// TwinCAT 3 PLC project SlaveController
// ProgramVersion: 3.1.4024.0
// libraries:
//   Tc2_EtherCAT, * (Beckhoff Automation GmbH)
//   Tc2_Math, * (Beckhoff Automation GmbH)
//   Tc2_Standard, * (Beckhoff Automation GmbH)
//   Tc2_System, * (Beckhoff Automation GmbH)
//   Tc2_Utilities, * (Beckhoff Automation GmbH)
//   Tc3_Module, * (Beckhoff Automation GmbH)
// project tree:
//   AgiMaths/Frames/ DHTrans.TcPOU (not stored), invFrame.TcPOU (not stored), rotX.TcPOU (not stored), rotY.TcPOU (not stored), rotZ.TcPOU (not stored), transform.TcPOU (not stored)
//   AgiMaths/MatrixLib/ angAxis2Rot.TcPOU (not stored), cross.TcPOU (not stored), Det5.TcPOU (not stored), Det6.TcPOU (not stored), Det7.TcPOU (not stored), invMat6.TcPOU (not stored), invMat6Old.TcPOU (not stored), invMat3.TcPOU (not stored), invMat7.TcPOU (not stored), Mat3T.TcPOU (not stored), matAdd.TcPOU (not stored), matMultiNum.TcPOU (not stored), matMultiply.TcPOU (not stored), matMultiVec.TcPOU (not stored), matSelfAdd.TcPOU (not stored), vecSelfAdd.TcPOU (not stored), matSelfSub.TcPOU (not stored), matSub.TcPOU (not stored), matTranspose.TcPOU (not stored), rot2AngAxis.TcPOU (not stored), vecAdd.TcPOU (not stored), norm.TcPOU (not stored), normalize.TcPOU (not stored), vecSelfMultiNum.TcPOU (not stored), vecMultiNum.TcPOU (not stored), vecSub.TcPOU (not stored)
//   AgiMaths/ sign.TcPOU (not stored), addVec7.TcPOU (not stored), atan2.TcPOU (not stored), cot.TcPOU (not stored)
//   DUTs/Enum/ E_CartJointState.TcTLEO (not stored), E_InstrumentType.TcDUT, E_MasterArmState.TcDUT (not stored), E_MatchedSlaveArmIdx.TcDUT (not stored), E_SetupArmState.TcDUT (not stored), E_SlaveArmState.TcDUT, E_DriverCtrlWord.TcDUT (not stored), E_DriverOPMode.TcDUT (not stored), E_DriverStatusWord.TcDUT
//   DUTs/Structure/MasterSlaveCommunication/ ST_MasterStatus.TcDUT, ST_SlaveStatus.TcDUT
//   DUTs/Structure/ ST_CartInputDataPool.TcDUT, ST_InstruOnChipData.TcDUT (not stored), ST_InstruStatus.TcDUT (not stored), ST_SetupArmCtrlCmds.TcDUT, ST_SetupInputDataPool.TcDUT, ST_SlaveArmCtrlCmds.TcDUT (not stored), ST_SlaveInputDataPool.TcDUT (not stored), ST_InstruKinematicParam.TcDUT, ST_Frame.TcDUT (not stored)
//   DUTs/Structure/TasksCommunication/ ST_CartJointData.TcDUT (not stored), ST_CartMotorInput.TcDUT (not stored), ST_CartMotorOutput.TcDUT (not stored), ST_CartUIData.TcDUT (not stored), ST_SetupStatus.TcDUT (not stored), ST_SetupJointData.TcDUT (not stored), ST_SlaveDynaData.TcDUT (not stored), ST_SlaveUIData.TcDUT (not stored), ST_CartStatus.TcDUT (not stored), ST_MasterJointData.TcDUT (not stored), ST_MotorInputs.TcDUT (not stored), ST_MotorOutputs.TcDUT (not stored), ST_SlaveJointData.TcDUT (not stored), ST_SafetyData.TcDUT
//   DUTs/Structure/UICommunication/ ST_cart_operation.TcDUT, ST_DH.TcDUT (not stored), ST_instrument_info.TcDUT (not stored), ST_scope_info.TcDUT, ST_state_machine_com.TcDUT (not stored), ST_ui_control.TcDUT (not stored)
//   DUTs/Type/ Mat34.TcDUT (not stored), Mat37.TcDUT (not stored), Mat43.TcDUT (not stored), Mat45.TcDUT (not stored), Mat4d.TcDUT (not stored), Mat5d.TcDUT (not stored), Mat67.TcDUT (not stored), Mat6d.TcDUT (not stored), Mat76.TcDUT (not stored), Mat7d.TcDUT (not stored), Vec2i.TcDUT, Vec4b.TcDUT (not stored), Vec4d.TcDUT (not stored), Vec4i.TcDUT (not stored), Vec5b.TcDUT (not stored), Vec5d.TcDUT (not stored), Vec5i.TcDUT (not stored), Vec6i.TcDUT (not stored), Vec8b.TcDUT (not stored), Vec8d.TcDUT (not stored), Vec8i.TcDUT (not stored), Mat3d.TcDUT (not stored), Vec3d.TcDUT (not stored), Vec6d.TcDUT (not stored), Vec7d.TcDUT (not stored), Vec7i.TcDUT (not stored)
//   FBs_Auxiliary/ FB_IOCheck.TcPOU (not stored), FB_IOToggleCheck.TcPOU (not stored), FB_rotaButtonDetect.TcPOU (not stored), FB_setupAdjustDetect.TcPOU, FB_setupJnt5AdjustDetect.TcPOU (not stored), FB_masterConnectionCheck.TcPOU (not stored), FB_trocarCheckDetect.TcPOU (not stored), FB_TrocarDetect.TcPOU, FB_PanelDetect.TcPOU, FB_InstrumentDetect.TcPOU, FB_AdjustDetect.TcPOU (not stored)
//   FBs_BasicControllers/ FB_dither.TcPOU (not stored), FB_InstrumentControl.TcPOU (not stored), FBMacroJntControl.TcPOU (not stored), FB_PID.TcPOU (not stored)
//   FBs_CartControlles/ FB_CartCtrlAdjust.TcPOU (not stored), FB_CartCtrlAsepticDeploy.TcPOU, FB_CartCtrlBase.TcPOU, FB_CartCtrlError.TcPOU, FB_CartCtrlInit.TcPOU (not stored), FB_CartCtrlInSurgery.TcPOU (not stored), FB_CartCtrlMotionCar.TcPOU (not stored), FB_CartCtrlReady.TcPOU, FB_CartCtrlRotaOverhang.TcPOU, FB_CartCtrlSlowDown.TcPOU, I_CartJointCtrl.TcIO
//   FBs_RobotDynamics/ FB_SlaveGravity.TcPOU, FB_SetupGravity.TcPOU
//   FBs_Robots/ FB_CartJoint.TcPOU (not stored), FB_CartRobot.TcPOU, FB_Instrument.TcPOU, FB_JointBase.TcPOU (not stored), FB_SlaveCart.TcPOU (not stored), FB_SetupArm.TcPOU (not stored), FB_SlaveJoint.TcPOU, FB_SetupJoint.TcPOU (not stored), FB_SetupRobot.TcPOU (not stored), FB_SlaveArm.TcPOU (not stored), FB_SlaveRobot.TcPOU (not stored)
//   FBs_SetupControllers/ FB_SetupCtrlDisable.TcPOU (not stored), FB_SetupCtrlJnt5GraCali.TcPOU, FB_SetupCtrlHold.TcPOU (not stored), FB_SetupCtrlManualAdjust.TcPOU, FB_SetupArmCtrlBase.TcPOU (not stored), FB_SetupCtrlAutoAdjust.TcPOU (not stored), FB_SetupCtrlCart.TcPOU (not stored), FB_SetupCtrlError.TcPOU (not stored), FB_SetupCtrlJnt3GraCali.TcPOU (not stored), FB_SetupCtrlInit.TcPOU (not stored), FB_SetupCtrlPackage.TcPOU (not stored), FB_SetupCtrlSelfCheck.TcPOU (not stored), I_SetupArmCtrl.TcIO (not stored)
//   FBs_SlaveControllers/ FB_SlaveCtrlDisable.TcPOU (not stored), FB_SlaveCtrlInstruInvasion.TcPOU, FB_SlaveCtrlInstruRetract.TcPOU (not stored), FB_SlaveCtrlInstruCali.TcPOU, FB_SlaveCtrlTest.TcPOU (not stored), FB_SlaveCtrlPackage.TcPOU (not stored), FB_SlaveCtrlEndoscope.TcPOU (not stored), FB_SlaveCtrlCart.TcPOU (not stored), FB_SlaveCtrlScopeReady.TcPOU (not stored), FB_SlaveCtrlSelfCheck.TcPOU (not stored), FB_SlaveCtrlError.TcPOU, FB_SlaveCtrlInstruReady.TcPOU (not stored), FB_SlaveCtrlMasterSlave.TcPOU (not stored), FB_SlaveCtrlMountInstru.TcPOU, FB_SlaveCtrlAdjust.TcPOU, FB_SlaveCtrlMountPanel.TcPOU (not stored), FB_SlaveCtrlPanelReady.TcPOU (not stored), FB_SlaveCtrlGraCali.TcPOU, FB_SlaveCtrlInit.TcPOU (not stored), FB_SlaveCtrlStandBy.TcPOU (not stored), FB_SlaveArmCtrlBase.TcPOU (not stored), I_SlaveArmCtrl.TcIO (not stored)
//   FBs_TrajectoryPlanning/ FB_BasicDoubleS.TcPOU (not stored), FB_trajBase.TcPOU (not stored), FB_TrajMoveJ.TcPOU (not stored), FB_setupTrajMoveJ.TcPOU (not stored), linear_trajectory_with_quintic_polynomial_blends.TcPOU (not stored), quintic_spline_curve.TcPOU (not stored), Quintic_spline_curve_factor.TcPOU (not stored), TrapezoIDal_velocity_trajectory.TcPOU (not stored)
//   FBs_TrajectoryPlanning/OTG/ FB_secOrdTrajFilter.TcPOU (not stored), FB_thirdOrdTrajFilter.TcPOU (not stored)
//   FBs_Filters/ FB_LowPassFilter.TcPOU (not stored)
//   GVLs/CartJoints/ GVL_CartControlParameters.TcGVL, GVL_CartJointEncoderCaliData.TcGVL, GVL_CartMotorParameters.TcGVL
//   GVLs/configs/robot3/ GVL_SetupArmDynamics_3.TcGVL (not stored), GVL_SlaveArmDynamics_3.TcGVL (not stored), GVL_SetupJointEncoderCaliData_3.TcGVL (not stored), GVL_SlaveJointEncoderCaliData_3.TcGVL
//   GVLs/configs/robot5/ GVL_SetupArmDynamics_5.TcGVL (not stored), GVL_SlaveArmDynamics_5.TcGVL, GVL_SetupJointEncoderCaliData_5.TcGVL (not stored), GVL_SlaveJointEncoderCaliData_5.TcGVL
//   GVLs/configs/robot4/ GVL_SetupArmDynamics_4.TcGVL (not stored), GVL_SetupJointEncoderCaliData_4.TcGVL, GVL_SlaveArmDynamics_4.TcGVL (not stored), GVL_SlaveJointEncoderCaliData_4.TcGVL (not stored)
//   GVLs/ GVL_CartParameters.TcGVL (not stored), GVL_com_upper_PC.TcGVL (not stored), GVL_InstruCtrlParams.TcGVL, GVL_MathDefine.TcGVL (not stored), GVL_SafetyParameters.TcGVL (not stored), GVL_SystemParameters.TcGVL (not stored)
//   GVLs/SetupArms/ GVL_SetupArmDynamics.TcGVL, GVL_SetupJointEncoderCaliData.TcGVL, GVL_SetupMotorParameters.TcGVL (not stored), GVL_SetupArmKinematic.TcGVL (not stored), GVL_SetupControlParameters.TcGVL (not stored)
//   GVLs/SlaveArms/ GVL_SlaveArmDynamics.TcGVL (not stored), GVL_SlaveArmKinematic.TcGVL (not stored), GVL_SlaveControlParameters.TcGVL, GVL_SlaveJointEncoderCaliData.TcGVL, GVL_SlaveMotorParameters.TcGVL (not stored)
//   Mains/ CartControl.TcPOU, SafetyCheck.TcPOU, SetupArmControl.TcPOU (not stored), SlaveArmControl.TcPOU (not stored), RobotDynamics.TcPOU (not stored)
//   SafetyCheck/ FB_CartCheck.TcPOU (not stored), FB_SetupArmCheck.TcPOU, FB_SlaveArmCheck.TcPOU (not stored)
//   / TaskCartControl.TcTTO (not stored), TaskDynamic.TcTTO (not stored), TaskSafetyCheck.TcTTO (not stored), TaskSetupArmControl.TcTTO (not stored), TaskSlaveArmControl.TcTTO (not stored)

// ---- DUTs/Enum/E_InstrumentType.TcDUT
TYPE E_InstrumentType :
(
	InstruType_UNKNOWM := 0,
	InstruType_CadiereForceps :=7,
	InstruType_NeedleDriver :=8,
	InstruType_MegaSCNeedleDriver :=9,// mega suture-cut needle driver
	InstruType_SCNeedleDriver :=10, // suture-cut needle driver
	InstruType_RoundTipScissors :=11,
	InstruType_ProGraspForceps :=12,
	InstruType_MarylandForceps :=13, // Maryland bipolar forceps
	InstruType_FenestratedForceps :=14, // Fnestrated bipolar forceps
	InstruType_CurvedScissors :=15, // monopolar curved scissors
	InstruType_CauteryHook :=16,
	InstruType_CauterySpatula :=17,
	InstruType_UltrasoundKnife :=18,
	InstruType_Endoscope := 20,
	InstruType_First := InstruType_CadiereForceps,
	InstruType_Last := InstruType_Endoscope
);
END_TYPE

// ---- DUTs/Enum/E_SlaveArmState.TcDUT
TYPE E_SlaveArmState :
(
	SlaveArmState_Error := 1,
	SlaveArmState_Init :=2,
	SlaveArmState_SelfCheck :=3,
	SlaveArmState_Standby :=4,
	SlaveArmState_MountPanel:=5,
	SlaveArmState_PanelReady :=6,
	SlaveArmState_MountInstru :=7,
	SlaveArmState_InstruReady :=8,
	SlaveArmState_MasterSlave :=9,
	SlaveArmState_ScopeReady :=10,
	SlaveArmState_EndoScope :=11,
	SlaveArmState_Adjust :=12,
	SlaveArmState_Package :=13,
	SlaveArmState_Cart := 14,
	SlaveArmState_GravityCali := 15,
	SlaveArmState_Test := 16,
	SlaveArmState_InstruRetract :=17,
	SlaveArmState_InstruInvasion :=18,
	SlaveArmState_Disable := 19,
	SlaveArmState_InstruCali := 20,
	
	SlaveArmState_totalNum :=SlaveArmState_InstruCali
);
END_TYPE

// ---- DUTs/Structure/MasterSlaveCommunication/ST_MasterStatus.TcDUT
// Input from master arm control task, including arm status and cartesian data
TYPE ST_MasterStatus :
STRUCT
	// master heart beat
	m_masterHeartBeat :INT:=0;
	
	// self-check trigger flag
	m_slaveSelfCheckFlag :BOOL :=FALSE;
	
	// linear motion scale
	m_motionScale : LREAL:=1.5;
	
	// state machine
	m_armState:ARRAY[1..g_mArmNum] OF E_masterArmState;
	
	// index(0 to 4) of slave arm which is tele-linked to master arm
	m_teleSlaveArmIdx :ARRAY[1..g_mArmNum] OF E_MatchedSlaveArmIdx;
	
	// grip angle
	m_gripAngle:ARRAY[1..g_mArmNum] OF LREAL;
	
	// current arm pose in monitor coordinate
	m_curArmPose:ARRAY[1..g_mArmNum] OF ST_Frame;
	
	// current arm twist[linear velocity; angular veloicty] in monitor coordinate
	m_curArmTwist:ARRAY[1..g_mArmNum] OF Vec6d;
	
END_STRUCT
END_TYPE

// ---- DUTs/Structure/MasterSlaveCommunication/ST_SlaveStatus.TcDUT
// Output from slave arm control task, including arm status and cartesian data
// Input to safety task and Master controller
TYPE ST_SlaveStatus :
STRUCT
	
	// state machine
	m_armState:ARRAY[1..g_sArmNum] OF E_SlaveArmState:=[g_sArmNum(SlaveArmState_Error)];
	
	// self-check pass flag
	m_selfCheckPass :ARRAY[1..g_sArmNum] OF BOOL :=[4(False)];
	
	// instrument info
	m_instruStauts :ARRAY[1..g_sArmNum] OF ST_InstruStatus;
	
	// flag if endoscope is mounted
	m_endoscopeMounted :BOOL := FALSE;
	
	// endoscope pose in cart coordinate
	m_endoscopePose : ST_Frame;
	
	// command arm pose in slave arm coordinate
	m_cmdArmPose:ARRAY[1..g_sArmNum] OF ST_Frame;
	
	// current arm pose in slave arm coordinate
	m_curArmPose:ARRAY[1..g_sArmNum] OF ST_Frame;
	
	// command arm twist[linear velocity; angular veloicty] in  slave arm coordinate
	m_cmdArmTwist:ARRAY[1..g_sArmNum] OF Vec6d;
	
	// current arm twist[linear velocity; angular veloicty] in  slave arm coordinate
	m_curArmTwist:ARRAY[1..g_sArmNum] OF vec6d;
	
	// master slave pose error [position, angle*axis] in endoscope coordinate
	m_masterSlavePoseError :ARRAY[1..g_sArmNum] OF Vec6d; 

END_STRUCT
END_TYPE

// ---- DUTs/Structure/ST_CartInputDataPool.TcDUT
TYPE ST_CartInputDataPool :
STRUCT
	// cart information, import from other task
	m_cartStatus AT %I*:ST_CartStatus;
	
	// safety information, import from safety check task
	m_safetyData AT %I*: ST_SafetyData;
	
	// slave status, import from slave control task
	m_slaveStatus AT %I*: ST_SlaveStatus;
	
	//UI information, import from UI controller
	m_UIData :ST_CartUIData;
	
	
END_STRUCT
END_TYPE

// ---- DUTs/Structure/ST_SetupArmCtrlCmds.TcDUT
TYPE ST_SetupArmCtrlCmds :
STRUCT
	// arm control data
	m_jntEnableFlag : Vec5i;
	m_jntOPMode : Vec5i;
	m_cmdJntPos : VEC5d;
	m_cmdJntVel : VEC5d;
	m_cmdJntAcc : VEC5d;
	m_cmdJntTrq : VEC5d;
	
END_STRUCT
END_TYPE

// ---- DUTs/Structure/ST_SetupInputDataPool.TcDUT
// Struct contains all data from other tasks and controller used for slave control
TYPE ST_SetupInputDataPool :
STRUCT
				
	// UI information, import from UI controller
	m_UIData AT %I*:ST_SlaveUIData;
	
	// slave status, import from slave control task
	m_slaveStatus AT %I*: ST_SlaveStatus;
	
	// safety information, import from safety check task
	m_safetyData AT %I*: ST_SafetyData;
	
	// cart information, import from other task
	m_cartStatus AT %I*:ST_CartStatus;
	
	// slave gravity
	m_setupJnt3Gravity AT %I* : ARRAY[1..g_sArmNum] OF LREAL;
	m_setupJnt5Gravity AT %I* :  ARRAY[1..g_sArmNum] of LREAL;
	
	
END_STRUCT
END_TYPE

// ---- DUTs/Structure/TasksCommunication/ST_SafetyData.TcDUT
// Output from safety check task
// Input to master arm control task
TYPE ST_SafetyData :
STRUCT
	m_slaveErrFlag :ARRAY[1..g_sArmNum] OF BOOL :=[4(FALSE)];
	m_setupErrFlag :ARRAY[1..g_sArmNum] OF BOOL :=[4(FALSE)];
	m_cartErrFlag :BOOL :=FALSE;
END_STRUCT
END_TYPE

// ---- DUTs/Structure/ST_InstruKinematicParam.TcDUT
 // instrumetn kinematic paramters
TYPE ST_InstruKinematicParam :
STRUCT	
	
	// instrument geometric parameters
	// NOTE: need update based on instrument types
	m_rodLength:LREAL:=0.5392;
	m_headLength:LREAL :=0.01;
	m_fingerLength:LREAL :=0;
	m_maxGripAngle :LREAL := 50.0 * g_deg2Rad;
	m_minGripAngle :LREAL := -25 * g_deg2Rad; // make sure fingers are fully closed
	
	// instrument kinematic parameters for joint/DH space transformation
	kx:lreal:=1;
	ky:lreal:=1;
	kz:LREAL:=1;
	k13:LREAL:=0.775;
	k23:LREAL:=0.775;
	m_openAngleDir:INT:=-1;
	
	// instrument wrist DH joint limit
	m_wristMinDHJntPos :Vec3d;
	m_wristMaxDHJntPos :Vec3d;

END_STRUCT
END_TYPE

// ---- DUTs/Structure/UICommunication/ST_cart_operation.TcDUT
TYPE ST_Cart_operation :
STRUCT
	Arm1_setup_sterile_state:UINT; //无菌袋安装完成，0：没有完成，1：完成
	Arm2_setup_sterile_state:UINT; //无菌袋安装完成，0：没有完成，1：完成
	Arm3_setup_sterile_state:UINT; //无菌袋安装完成，0：没有完成，1：完成
	Arm4_setup_sterile_state:UINT; //无菌袋安装完成，0：没有完成，1：完成
	
	draping_posture_state:UINT; //姿态调整状态，0：没有完成，1：完成
	setup_sterile_state:UINT; //无菌袋安装完成，0：没有完成，1：完成
	docking_posture_state:UINT; //姿态调整状态，0：没有完成，1：完成
	
	//Cart_move_to_sterile_state:UINT; //台车移动到无菌区粗摆位，0：没有完成，1：完成
	Cart_static_in_sterile_state:UINT; //台车进入无菌区，并且台车停止运动(连续10s没有运动)，0：没有完成，1：完成
	
	//scope_adapter_install_state:UINT; //腔镜转接头卡接完成，0：没有完成，1：完成	
	scope_install_state:UINT; //腔镜卡接完成
	//scope_fixed_point_confirm:UINT; //腔镜不动点确认完成
	
	//surgical_posture_adjust:UINT; //台车中调整
	all_fixed_point_confirm:UINT; //所有不动点确定---手术中的标志
	//all_fixed_point_unlock:UINT; //所有不动点解锁---手术结束标志（所有无菌袋拿掉）
	stow_posture_state:UINT; //所有机械臂收纳完成
END_STRUCT
END_TYPE

// ---- DUTs/Structure/UICommunication/ST_scope_info.TcDUT
TYPE ST_scope_info :
STRUCT
	is_connected:BOOL;
	is_ready:BOOL;
	id:UINT;
	scope_deg:UINT;
	scope_up_down:UINT;
	scope_gravity_angle:INT;
	scope_name:STRING;
END_STRUCT
END_TYPE

// ---- DUTs/Type/Vec2i.TcDUT
TYPE Vec2i : ARRAY[1..2] OF INT; END_TYPE

// ---- DUTs/Enum/E_DriverStatusWord.TcDUT
TYPE E_DriverStatusWord :
(
	DriverStatusWord_INIT := 4641,
	DriverStatusWord_PREOP := 4659,
	DriverStatusWord_OP := 4663,
	
	MZDriverStatusWord_SwitchOnDisable := 16#40,
	MZDriverStatusWord_ReadyToSwitchOn := 16#21,
	MZDriverStatusWord_SwitchOn := 16#33,
	MZDriverStatusWord_OperationEnbale := 16#37,
	MZDriverStatusWord_Fault := 16#08
);
END_TYPE

// ---- GVLs/CartJoints/GVL_CartControlParameters.TcGVL
{attribute 'global_init_slot' := '49991'} 
{attribute 'qualified_only'}
VAR_GLOBAL
	// filter cut-off frequency for velocity and torque
	g_curJntVelLpfCutoffFreq :LREAL := 30;
	g_cmdJntTrqLpfCutoffFreq :LREAL := 300;
	g_curJntTrqLpfCutoffFreq :LREAL := 300;
	
	g_curBeamStretchJntInitPos :LREAL := 0.972;
	g_maxCartVel :ARRAY [1..4] OF LREAL:= [0.016, 0.05, 0.05, 0.05];
	
	g_maxJntVel :ARRAY [1..8] OF LREAL:=[0.0025, 0.0025, 2.3, 2.3, 0.016, 5*g_deg2Rad, 0.050, 5*g_deg2Rad];
	g_maxJntAcc :ARRAY [1..8] OF LREAL:=[0.0025*2, 0.0025*2, 2.3*2, 2.3*2, 0.016*2, 5*g_deg2Rad*2, 0.050*2, 5*g_deg2Rad*2];
	
	g_surgicalOrientPos : ARRAY [1..5, 1..3, 1..4]  OF LREAL := [
		0.1, 0.10, 0.10, 0.10,    0.1, -0.10, 0.10, -0.10,	0.1, 0.10, 0.10, -0.10,
		0.2, 0.20, 0.20, 0.20,    0.2, -0.20, 0.20, -0.20,	0.2, 0.20, 0.20, -0.20,
		0.3, 0.25, 0.30, 0.30,    0.3, -0.25, 0.30, -0.30,	0.3, 0.25, 0.30, -0.30,
		0.4, 0.30, 0.35, 0.35,    0.4, -0.30, 0.35, -0.35,	0.4, 0.30, 0.35, -0.35,
		0.5, 0.35, 0.40, 0.40,    0.5, -0.35, 0.40, -0.40,	0.4, 0.30, 0.35, -0.35];
	
	g_surgicalDrapingPos : ARRAY[1..8] OF LREAL := [0, 0, 0, 0, 0.3, 0, 0.2, 0];
	
	g_jntCtrlAngTolHigh :LREAL :=1*g_deg2Rad;
END_VAR

// ---- GVLs/CartJoints/GVL_CartJointEncoderCaliData.TcGVL
{attribute 'qualified_only'}
// Robot5 --joints parameters of setup arms
VAR_GLOBAL
	// absolute encoder value at minimal joint positon
	g_minLinkEncoder :ARRAY[1..g_cartJntNum] OF DINT :=[0, 0, 0, 0, 39509461, 14558528, 57761547, 8171292];
		 
	// absolute encoder value at maximum joint positon
	g_maxLinkEncoder :ARRAY[1..g_cartJntNum] OF DINT :=[0, 0, 0, 0, 36724181, 577308, 59809539,7327520 ];
	
	// absolute encoder value at calibrated positon
	g_caliLinkEncoder :ARRAY[1..g_cartJntNum] OF DINT :=[0, 0, 0, 0, 39509461, 15956526, 59809539, 16172652];
	
	 // if absolute encoder value cross zeros within joint motion range
	g_linkEncZeroCross :ARRAY[1..g_cartJntNum] OF INT :=[0, 0, 0, 0, 0, 1, 0, 1];
		 

	// abolute encoder expanded limit buffer in case there is calibrtion error at limit position
	g_linkEncLimitBuffer : DINT := 100000;

	// absolute encoder direction
	g_asbEncoderDir :ARRAY[1..g_cartJntNum] OF INT :=[1, 1, 1, 1, -1, 1, -1, -1];
													
	// flag if joint can rotate multiple cycles
	g_multipleCyclesJoint :ARRAY[1..g_cartJntNum] OF INT :=[0, 0, 0, 0, 0, 0, 0, 0];
		 
	// joint position at link encoder calibrated point
	g_linkEncCaliJntPos :ARRAY[1..g_cartJntNum] OF LREAL :=[0.0, 0.0, 0.0, 0.0, 0.0, 0.0, 0, 0.0];
	
	 // joint SDO address
	g_slaveCartNetID: T_AmsNetId:='169.254.186.39.7.1';
	g_slaveCartJointNetPort:ARRAY[1..g_cartJntNum] OF UINT :=[1005,	1004,	1003,	1002,	1001,   1006,  1007,  1008];

END_VAR

// ---- GVLs/CartJoints/GVL_CartMotorParameters.TcGVL
{attribute 'global_init_slot' := '49991'}
{attribute 'qualified_only'}
VAR_GLOBAL CONSTANT
	// encoder resolution
	//TODO: resolution of joint 2/3 need verification
	g_incEncoderRes :ARRAY[1..g_cartJntNum] OF DINT :=[2(65536), 4*2500, 4*2500, 4*2500, 3(65536)];
	g_absEncoderRes :ARRAY[1..g_cartJntNum] OF DINT :=[1, 1, 1, 1, 8192, 16777215, 8192,16777215];
	
	// reduction ratio
	g_motorReduction :ARRAY[1..g_cartJntNum] OF LREAL :=
		[100.75*2*pi/0.002, 100.75*2*pi/0.002, 160, 160, 
		 5*(2*pi)/0.005, 676.0/49*356, 299.0/14*(2*pi)/0.020, 676.0/49*238];
	g_absEncoderReduction :ARRAY[1..g_cartJntNum] OF LREAL :=[4(1.0), 2*pi/0.002 , 1.0, 2*pi/0.002, 1.0];
	 
	// motor parameters
	g_motorTrqConst :ARRAY[1..g_cartJntNum] OF LREAL :=[ 0.0256, 0.0256, 0.058,0.058,  0.123,0.0292,0.0292,0.0292];
	g_motorMaxCurrent :ARRAY[1..g_cartJntNum] OF LREAL :=[ 41200,41200,50000,50000,  33000,41200,41200,41200];//mA
	
	// motor and absEncoder direction
	g_motorDir :ARRAY[1..g_cartJntNum] OF INT :=[1, 1, 1, 1, 1, 1, -1, -1];
																												 
	// joint position limit
	g_minJntPos: ARRAY[1..g_cartJntNum] OF LREAL:=[0, 0, 1, 1, 0, -30*g_deg2Rad, 0.002, -160*g_deg2Rad];	
	g_maxJntPos: ARRAY[1..g_cartJntNum] OF LREAL:=[0.053, 0.053, 1, 1,  0.6, 30*g_deg2Rad, 0.498, 160*g_deg2Rad];	
	
	// joint velocity limit
	g_maxJntVel :ARRAY[1..g_cartJntNum] OF LREAL :=[0.0025, 0.0025, 2.3, 2.3, 0.016, 5*g_deg2Rad, 0.050*g_deg2Rad, 5*g_deg2Rad];
	g_maxJntAcc :ARRAY[1..g_cartJntNum] OF LREAL :=[0.0025 * 2, 0.0025 * 2, 2.3 * 2, 2.3 * 2, 0.016 * 2, 5*g_deg2Rad * 2, 0.050*g_deg2Rad * 2, 5*g_deg2Rad * 2];
END_VAR

// ---- GVLs/configs/robot3/GVL_SlaveJointEncoderCaliData_3.TcGVL
{attribute 'qualified_only'}
// Robot3 --joints parameters of slave arms
VAR_GLOBAL CONSTANT	
	// absolute encoder value at minimal joint positon
	g_minLinkEncoder :ARRAY[1..g_sArmNum, 1..g_sJntNum] OF DINT :=
		[796618, 12395160, 5368016, 0, 0, 0, 0, 0,
		 13317378, 3888760, 9175760, 0, 0, 0, 0, 0,
		 823964, 3955316, 15205696, 0, 0, 0, 0, 0,
		 4820816, 7977020, 9226720, 0, 0, 0, 0, 0];
		 
	// absolute encoder value at maximum joint positon
	g_maxLinkEncoder :ARRAY[1..g_sArmNum, 1..g_sJntNum] OF DINT :=
		[15464922, 5123844, 14570432, 0, 0, 0, 0, 0,
		 11230582, 13464106, 1613344, 0, 0, 0, 0, 0,
		 15526052, 13536910, 7701984, 0, 0, 0, 0, 0,
		 2731020, 789080, 1671808, 0, 0, 0, 0, 0];
	
	// absolute encoder value at calibrated positon
	g_caliLinkEncoder :ARRAY[1..g_sArmNum, 1..g_sJntNum] OF DINT :=
		[8162412, 8169482, 14570432, 15377856,15482848, 7058832, 6935120, 7155184,
		 3932766, 16478880, 1613344, 15324752, 15485488, 7135776, 7032592, 6946704,
		 8248074, 16595424, 7701984, 15349408, 15361392, 6997280, 6757296, 720176,
		 12196142, 3807946, 1671808, 15274368, 15387696, 6812992, 6747792, 13454432];
	
	 // if absolute encoder value cross zeros within joint motion range
	 // NOTICE: joint 7 is always 0.
	g_linkEncZeroCross :ARRAY[1..g_sArmNum, 1..g_sJntNum] OF INT :=
		[0, 0, 0, 1, 1, 1, 1, 1,
		 1, 1, 1, 1, 1, 1, 1, 1,
		 0, 1, 1, 1, 1, 1, 1, 1,
		 1, 0, 1, 1, 1, 1, 1, 1];
		 
	 // joint SDO address
	g_slaveArmNetID: ARRAY[1..4] OF T_AmsNetId:=['169.254.186.39.3.1','169.254.186.39.8.1','169.254.186.39.9.1','169.254.186.39.10.1'];
	g_slaveJointNetPort:ARRAY[1..g_sArmNum,1..g_sJntNum] OF UINT :=[
		1006,	1007,	1008,	2(1009),	3(1010),
		1006,	1007,	1008,	2(1009),	3(1010),
		1006,	1007,	1008,	2(1009),	3(1010),
		1006,	1007,	1008,	2(1009),	3(1010)];
		
//################ DO NOT modify parameters below ###########################
	// abolute encoder expanded limit buffer in case there is calibrtion error at limit position
	g_linkEncLimitBuffer : DINT := 100000;
	
	// absolute encoder direction
	g_asbEncoderDir :ARRAY[1..g_sJntNum] OF INT :=[1, -1, 1, 1, 1, 1, 1, 1];
	
	// flag if joint can rotate multiple cycles
	g_multipleCyclesJoint :ARRAY[1..g_sArmNum, 1..g_sJntNum] OF INT :=
		[0, 0, 0, 1, 1, 1, 1, 1,
		 0, 0, 0, 1, 1, 1, 1, 1,
		 0, 0, 0, 1, 1, 1, 1, 1,
		 0, 0, 0, 1, 1, 1, 1, 1];
		 
	// joint position at link encoder calibrated point
	g_linkEncCaliJntPos :ARRAY[1..g_sJntNum] OF LREAL :=
		[0.0, -PI/2, 0.581633, 5(0.0)];

	
END_VAR

// ---- GVLs/configs/robot5/GVL_SlaveArmDynamics_5.TcGVL
{attribute 'global_init_slot' := '49992'}
{attribute 'qualified_only'}
// Robot5 --dynamic parameters of slave arms
VAR_GLOBAL CONSTANT
	
(*graParam=[ 9.8*m5,...
           0.41601*m2 + 0.41601*m3 + 0.0000216012*m4 + 0.0000216012*m5 + 9.8*mx1 - 1.3639*mx3 - 9.70463*my3,...
           9.8*mz2 - 9.8*my5 - 9.8*my1 + 9.8*mz3 + 9.8*mz4,...
           2.19651*m3 + 2.19651*m4 + 0.00000258969*m5 + 8.64766*mx2 - 4.61063*my2 + 9.8*my4 + 9.8*mz5,...
          1.1711*m3 + 1.1711*m4 + 0.00000122416*m5 + 4.61063*mx2 - 9.8*mx4 - 9.8*mx5 + 8.64766*my2]'
*)			
	// robot No.4
	g_gravityParam :ARRAY[1..4,1..5] OF REAL := 
	[ 7.5951,    1.6336,   -4.2417,    9.4106,    4.7289,
	  7.4741,    3.7472,   -4.4567,   10.5517,    7.6095,
	  7.6732,    3.7472,   -4.4458,    9.6721,    7.2742,
	  7.4582,    3.5688,   -3.7215,    9.2746,    5.7641];
	 
	g_gravityTrocar :ARRAY[1..5] OF REAL :=[0.1661, -0.4124,  0.0964,   -0.7987,   -0.6999 ];
	g_gravityInstrument :ARRAY[1..5] OF REAL :=[ 3.1217,  -0.3099,   0.0778,   -1.2498,   -0.8041];
	g_gravityEndoscope :ARRAY[1..5] OF REAL :=[10.8619,  -0.8575,   -1.0274,   -0.2425,   -0.0869];
	
	// joint friction(with instrument mounted)
	g_slaveJntFriction :ARRAY[1..g_sArmNum, 1..g_sJntNum] OF LREAL :=
			[ 5.3354,    9.5437,    4.6271,  0.03, 0.03, 0.03, 0.03, 0,
			  4.5927,    9.6040,    3.7367, 0.03, 0.03, 0.03, 0,
		      4.3557,    8.4286,    5.9078,  0.03, 0.03, 0.03, 0.03, 0,
              4.1447,    7.2202,    6.8253,  0.03, 0.03, 0.03, 0.03, 0	 ];
	
END_VAR

// ---- GVLs/configs/robot5/GVL_SlaveJointEncoderCaliData_5.TcGVL
{attribute 'qualified_only'}
// Robot5 --joints parameters of slave arms
VAR_GLOBAL CONSTANT
	// absolute encoder value at minimal joint positon
	g_minLinkEncoder :ARRAY[1..g_sArmNum, 1..g_sJntNum] OF DINT :=
		[13299286, 12259316, 8131200, 0, 0, 0, 0, 0,
		 7690928, 8194684, 1783424, 0, 0, 0, 0, 0,
		 13300276, 12243976, 15232032, 0, 0, 0, 0, 0,
		 752828, 16341268, 3536512, 0, 0, 0, 0, 0];
		 
	// absolute encoder value at maximum joint positon
	g_maxLinkEncoder :ARRAY[1..g_sArmNum, 1..g_sJntNum] OF DINT :=
		[11218724, 5032692, 509984, 0, 0, 0, 0, 0,
		 15388748, 943300, 10993024, 0, 0, 0, 0, 0,
		 11204586, 5012744, 7690928, 0, 0, 0, 0, 0,
		 15415998, 9127988, 12720912, 0, 0, 0, 0, 0];
	
	// absolute encoder value at calibrated positon
	g_caliLinkEncoder :ARRAY[1..g_sArmNum, 1..g_sJntNum] OF DINT :=
		[3882398, 8083626, 509984, 13079328, 101984, 14934512, 4402512, 5578752,
		 8049042, 3955388, 10993024, 15376976, 15429216, 6997360, 7093456, 7154688,
		 3865836, 8052426, 7690928, 15280848, 15470720, 7024336, 7061984, 7187520,
		 8117082, 12176494, 12720912, 15362624, 15519280, 6971776, 6970208, 7079008];
	
	 // if absolute encoder value cross zeros within joint motion range
	 // NOTICE: joint 7 is always 0.
	g_linkEncZeroCross :ARRAY[1..g_sArmNum, 1..g_sJntNum] OF INT :=
		[1, 0, 1, 1, 1, 1, 1, 1,
		 0, 0, 0, 1, 1, 1, 1, 1,
		 1, 0, 1, 1, 1, 1, 1, 1,
		 0, 0, 0, 1, 1, 1, 1, 1];
		 
	 // joint SDO address
	g_slaveArmNetID: ARRAY[1..4] OF T_AmsNetId:=['169.254.186.39.3.1','169.254.186.39.8.1','169.254.186.39.9.1','169.254.186.39.10.1'];
	g_slaveJointNetPort:ARRAY[1..g_sArmNum,1..g_sJntNum] OF UINT :=[
		1006,	1007,	1008,	2(1009),	3(1010),
		1006,	1007,	1008,	2(1009),	3(1010),
		1006,	1007,	1008,	2(1009),	3(1010),
		1006,	1007,	1008,	2(1009),	3(1010)];
		
//################ DO NOT modify parameters below ###########################
	// abolute encoder expanded limit buffer in case there is calibrtion error at limit position
	g_linkEncLimitBuffer : DINT := 100000;
	
	// absolute encoder direction
	g_asbEncoderDir :ARRAY[1..g_sJntNum] OF INT :=[1, -1, 1, 1, 1, 1, 1, 1];
	
	// flag if joint can rotate multiple cycles
	g_multipleCyclesJoint :ARRAY[1..g_sArmNum, 1..g_sJntNum] OF INT :=
		[0, 0, 0, 1, 1, 1, 1, 1,
		 0, 0, 0, 1, 1, 1, 1, 1,
		 0, 0, 0, 1, 1, 1, 1, 1,
		 0, 0, 0, 1, 1, 1, 1, 1];
		 
	// joint position at link encoder calibrated point
	g_linkEncCaliJntPos :ARRAY[1..g_sJntNum] OF LREAL :=
		[0.0, -PI/2, 0.581633, 5(0.0)];

	
END_VAR

// ---- GVLs/configs/robot4/GVL_SetupJointEncoderCaliData_4.TcGVL
{attribute 'qualified_only'}
// Robot4 --joints parameters of setup arms
VAR_GLOBAL
	// absolute encoder value at minimal joint positon
	g_minLinkEncoder :ARRAY[1..g_sArmNum, 1..g_setupJntNum] OF DINT :=
		[3491080, 45629648, 37611523, 14466480, 9529300,
		 11218068, 40471181, 46688105, 1920038, 1149668,
		 13090440, 42200874, 47769403, 1835700, 9556586,
		 3185760, 43906815, 38691136, 1756138, 5310180];
		 
	// absolute encoder value at maximum joint positon
	g_maxLinkEncoder :ARRAY[1..g_sArmNum, 1..g_setupJntNum] OF DINT :=
		[15549460, 44184373, 36803146, 12923670, 757636,
		 6485500, 39023966, 45894528, 350598, 9152796,
		 8418056, 40752101, 46971620, 296506, 778048,
		 15218140, 42459588, 37898741, 213910, 13319010];
	
	// absolute encoder value at calibrated positon
	g_caliLinkEncoder :ARRAY[1..g_sArmNum, 1..g_setupJntNum] OF DINT :=
		[1118980, 44184373, 37611523, 5005500, 5136494,
		 8825840, 39023966, 46688105, 9194020, 13570056,
		 10746684, 40752101, 47769403, 9121174, 5171970,
		 813364, 42459588, 38691136, 9153890, 934780];
	
	 // if absolute encoder value cross zeros within joint motion range
	g_linkEncZeroCross :ARRAY[1..g_sArmNum, 1..g_setupJntNum] OF INT :=
		[1, 0, 0, 1, 0,
		 0, 0, 0, 1, 1,
		 0, 0, 0, 1, 0,
		 1, 0, 0, 1, 1];
		 
//################ DO NOT modify parameters below ###########################
	// abolute encoder expanded limit buffer in case there is calibrtion error at limit position
	g_linkEncLimitBuffer : DINT := 100000;

	// absolute encoder direction
	g_asbEncoderDir :ARRAY[1..g_setupJntNum] OF INT :=[-1, -1, -1, 1, -1];
													
	// flag if joint can rotate multiple cycles
	g_multipleCyclesJoint :ARRAY[1..g_sArmNum, 1..g_setupJntNum] OF INT :=
		[0, 0, 0, 0, 0,
		 0, 0, 0, 0, 0,
		 0, 0, 0, 0, 0,
		 0, 0, 0, 0, 0];
		 
	// joint position at link encoder calibrated point
	g_linkEncCaliJntPos :ARRAY[1..g_sArmNum, 1..g_setupJntNum] OF LREAL :=
		[-140*g_deg2Rad, 0.779, 0.0, 90.0*g_deg2Rad, 0.0,
		 -115*g_deg2Rad, 0.607, 0.0, 90.0*g_deg2Rad, 0.0,
		 -65*g_deg2Rad, 0.607, 0.0, 90.0*g_deg2Rad, 0.0,
 		 -40*g_deg2Rad, 0.779, 0.0, 90.0*g_deg2Rad, 0.0];
	

END_VAR

// ---- GVLs/GVL_InstruCtrlParams.TcGVL
// TODO： Code review and refined
VAR_GLOBAL
	
	//器械相关
	Head_Len_1:ARRAY[1..30] OF LREAL:=[1,1,1,1,1,1,	0.01950, 0.0096, 0.0109, 0.011,		0.01101, 0.02313, 0.0195, 0.0207, 0.0130, 0.01638, 0.01638, 13(1)	];
	
	camera_slope_angle:LREAL:=30.0*g_deg2Rad;; //摄像头斜面角度
	
	a3:ARRAY[1..30] OF LREAL:=[1,1,1,1,1,1,  0.0089,0.0089,0.010,0.010,		0.0089,0.01065,0.01065,0.01065,0.0089,		0.00935,0.00935,0,0,   4(0), 0.0089, 5(0)];
	k13:ARRAY[1..30] OF LREAL:=[1,1,1,1,1,1, 0.77510204, 0.808510638, 0.62295082, 0.644067797,  0.729166667,  0.5, 0.62295082, 0.62295082,  0.729166667,   -0.734693878,	-0.734693878,    1,      1,   1,	4(1), 0.77510204, 5(1)];
	k23:ARRAY[1..30] OF LREAL:=[1,1,1,1,1,1, 0.77510204, 0.808510638, 0.62295082, 0.644067797,  0.729166667,  0.5, 0.62295082, 0.62295082,  0.729166667,   -0.734693878,	-0.734693878,    1,      1,   1,	4(1), 0.77510204, 5(1)  ];
	kx:ARRAY[1..30] OF LREAL:=[30(-1)];
	ky:ARRAY[1..30] OF LREAL:=[1,1,1,1,1,1,  0.931034483,    0.931034483,      0.931034483,    0.931034483,    0.947368421,    0.931034483,    0.931034483,     0.931034483,     0.931034483,   0.877192982,	0.877192982,    1,      1,   1,	4(1), 0.931034483, 5(1)   ];
	kz:ARRAY[1..30] OF LREAL:=[1,1,1,1,1,1,  0.844827586,    0.810344828,      1.051724138,    1.017241379,    0.842105263,    1.310344828,    1.051724138,     1.051724138,     0.827586207,   0.859649123,	0.859649123,    1,      1,   1,	4(1), 0.844827586, 5(1)  ];
	openAngleDir:ARRAY[1..30] OF INT:=[30(-1)];
	
	rad_30:LREAL:=30.0*g_deg2Rad;  rad_60:LREAL:=60.0*g_deg2Rad;	 rad_38:LREAL:=38.0*g_deg2Rad;	rad_55:LREAL:=55.0*g_deg2Rad;	
	rad_45:LREAL:=45.0*g_deg2Rad; rad_28:LREAL:=28.0*g_deg2Rad; rad_10:LREAL:=10.0*g_deg2Rad;rad_90:LREAL:=90.0*g_deg2Rad;
	open_angle_max:ARRAY[1..30] OF LREAL:=[1,1,1,1,1,1,  rad_45,  rad_30+rad_10,  rad_38+rad_10, rad_38+rad_10,	 rad_30+rad_10, rad_90, rad_45+rad_10, rad_45+rad_10,  rad_60,rad_30,     rad_30,1,1];
	
	tool_name:ARRAY[1..30] OF STRING:=['1','1','1','1','1','1',  'Cadiere Forceps','Large Needle Driver','Mega SutureCut Needle Driver','Large SutureCut Needle Driver',	'RoundTip Scissors','Prograsp',	'Maryland Bipolar Forceps','Fenestrated Bipolar Forceps', 'Monopolar Curved Scissors','Permanent Cautery Hook','Permanent Cautery Spatula','Ultrasound Knife','1','Camera'];
	
//	Head_Len:ARRAY[1..30] OF LREAL:=[1,1,1,1,1,1,	0.01950, 0.0096, 0.0109, 0.011,		0.01101, 0.02313, 0.0195, 0.0207, 0.0130, 0.01638, 0.01638, 13(1)	];
	Head_Len:ARRAY[1..30] OF LREAL:=[0,0,0,0,0,0,	0, 0.0096, 0.0109,  0.0109,		0, 0, 0, 0, 0, 0, 0, 13(0)	];
		
	//*************************绝对定位精度测试使用*****************************//
	len1:LREAL:=0.5438;  len3:LREAL:=0.009;	len_camera:LREAL:=0.49;//0.477;//0.3035;//0.51	
	Len_Rod:ARRAY[1..30] OF LREAL:=[0,0,0,0,0,  0, len1,len1,len1,len1,	len1,len1,len1,len1,0.54375,	0.5432, 0.5432,0,0,len_camera,     4(0),0.551,5(0)]; //器械的杆长	，ID25号器械是主从延时测试用，长度为533+18
	
	Len_mounting_surface:ARRAY[1..30] OF LREAL:=[0,0,0,0,0,	0,len3,len3,len3,len3,	len3,len3,len3,len3,len3,	len3,len3,0,0,len3,    4(0),len3,5(0)]; //滑块和器械安装面的距离(图中的L3)
	TroCar_Len:LREAL:=0.1;//穿刺器长度、此处使用的是短穿刺器
	Zero_To_Bottom_J8:LREAL:=0.14;//8关节刻度线到最底部长度

	// master gripper angle limit
	g_maxMasterGripAngle :LREAL := 30*g_deg2Rad;
	g_minMasterGripAngle : LREAL :=0.0;
	g_masterGripForceStartAng :LREAL :=5*g_deg2Rad;
	
	//ultrasound knife kinematics parameter
	g_uknifeGripTravel :LREAL:= 0.00353;
	g_uknifeGripDividAngle : LREAL := 17 * g_deg2Rad;
	g_uknifeMotorLead : LREAL := 0.025;
	g_uknifeLeverRatio : LREAL := 13.0/18.5;
	
	
	
	
END_VAR

// ---- GVLs/SetupArms/GVL_SetupArmDynamics.TcGVL
{attribute 'global_init_slot' := '49992'}
{attribute 'qualified_only'}
// Robot5 --dynamic parameters of setup arms
VAR_GLOBAL 
	(* setup joint5 gravity parameters. last 5 parameters are defined in slave arm dynamic
	% graParam=[ 9.8*mx0,...
	%            4.92539*m1 + 4.92539*m2 + 4.92539*m3 + 7.8853*m4 + 7.8853*m5 + 9.70463*mx3 - 9.8*my0 - 1.3639*my3 + 9.8*mz1,...
	%            9.8*m5,...
	%            0.41601*m2 + 0.41601*m3 + 0.0000216012*m4 + 0.0000216012*m5 + 9.8*mx1 - 1.3639*mx3 - 9.70463*my3,...
	%            9.8*mz2 - 9.8*my5 - 9.8*my1 + 9.8*mz3 + 9.8*mz4,...
	%            2.19651*m3 + 2.19651*m4 + 0.00000258969*m5 + 8.64766*mx2 - 4.61063*my2 + 9.8*my4 + 9.8*mz5,...
	%            1.1711*m3 + 1.1711*m4 + 0.00000122416*m5 + 4.61063*mx2 - 9.8*mx4 - 9.8*mx5 + 8.64766*my2]';
	*)				
	//setup joint5 gravity parameters
	g_setupJnt5GravityParam :ARRAY[1..4,1..2] OF REAL := 
	[ 0.0000,   54.4806,
	  0.0196,   61.5623,
	  0.0196,   65.0026,
	  0.0196,   59.3080 ];

	(* setup joint3 gravity parameters
	 graParams = [p1,p2,p3,p4]
	 gravity = p1*q^3 + p2*q^2 + p3^q + p4
	 q(- [q0,q1]*)
 	// setup joint3 gravity parameter
	g_setupJnt3GravityParams :ARRAY[1..4, 1..4] OF LREAL :=
	[ 12732.1, -2686.58, 277.075, -95.1403,
	 -4213.4, 1194.4, 207.745, -118.926,
	3798.81, -862.596, 397.288, -127.846,
	 35991.5, -10457.4, 1058.33, -122.463];
	 
	(* setup joint3 friction parameters
	 graParams = [p1mp2,p3,p4]
	 friciton = p1*q^3 + p2*q^2 + p3^q + p4
	 q(- [q0,q1]*)
 	// setup joint3 friction parameter
	g_setupJnt3FrictionParams :ARRAY[1..4, 1..4] OF LREAL :=
	[  -41668.6, 14453.2, -1563.43, 100.562,
	 -16563.6, 8089.53, -1307.53, 112.977,
	-39448.5, 15129.4, -1976.17, 137.28,
	-26846.1, 9145.03, -1006.01, 79.1108];
	
	g_setupJnt3GravityPosRange :ARRAY[1..4, 1..2] OF REAL :=
	[ 0.0189,    0.1788,
	  0.0189,    0.1790,
	  0.0188,    0.1788,
	  0.0188,    0.1788];
 	
	 
	// joint gravity offset
	g_setupJntGravityOffset :ARRAY[1..4,1..5] OF REAL := 
	[0, 0, 0, 0,  0,
	 0, 0, 0, 0,  0,
	 0, 0, 0, 0,  0,
	 0, 0, 0, 0,  0];

END_VAR

// ---- GVLs/SetupArms/GVL_SetupJointEncoderCaliData.TcGVL
{attribute 'qualified_only'}
// Robot4 --joints parameters of setup arms
VAR_GLOBAL
	// absolute encoder value at minimal joint positon
	g_minLinkEncoder :ARRAY[1..g_sArmNum, 1..g_setupJntNum] OF DINT :=
		[3491080, 45629648, 37611523, 14466480, 9529300,
		 11218068, 40471181, 46688105, 1920038, 1149668,
		 13090440, 42200874, 47769403, 1835700, 9556586,
		 3185760, 43906815, 38691136, 1756138, 5310180];
		 
	// absolute encoder value at maximum joint positon
	g_maxLinkEncoder :ARRAY[1..g_sArmNum, 1..g_setupJntNum] OF DINT :=
		[15549460, 44184373, 36803146, 12923670, 757636,
		 6485500, 39023966, 45894528, 350598, 9152796,
		 8418056, 40752101, 46971620, 296506, 778048,
		 15218140, 42459588, 37898741, 213910, 13319010];
	
	// absolute encoder value at calibrated positon
	g_caliLinkEncoder :ARRAY[1..g_sArmNum, 1..g_setupJntNum] OF DINT :=
		[1118980, 44184373, 37611523, 5005500, 5136494,
		 8825840, 39023966, 46688105, 9194020, 13570056,
		 10746684, 40752101, 47769403, 9121174, 5171970,
		 813364, 42459588, 38691136, 9153890, 934780];
	
	 // if absolute encoder value cross zeros within joint motion range
	g_linkEncZeroCross :ARRAY[1..g_sArmNum, 1..g_setupJntNum] OF INT :=
		[1, 0, 0, 1, 0,
		 0, 0, 0, 1, 1,
		 0, 0, 0, 1, 0,
		 1, 0, 0, 1, 1];
		 
//################ DO NOT modify parameters below ###########################
	// abolute encoder expanded limit buffer in case there is calibrtion error at limit position
	g_linkEncLimitBuffer : DINT := 100000;

	// absolute encoder direction
	g_asbEncoderDir :ARRAY[1..g_setupJntNum] OF INT :=[-1, -1, -1, 1, -1];
													
	// flag if joint can rotate multiple cycles
	g_multipleCyclesJoint :ARRAY[1..g_sArmNum, 1..g_setupJntNum] OF INT :=
		[0, 0, 0, 0, 0,
		 0, 0, 0, 0, 0,
		 0, 0, 0, 0, 0,
		 0, 0, 0, 0, 0];
		 
	// joint position at link encoder calibrated point
	g_linkEncCaliJntPos :ARRAY[1..g_sArmNum, 1..g_setupJntNum] OF LREAL :=
		[-140*g_deg2Rad, 0.779, 0.0, 90.0*g_deg2Rad, 0.0,
		 -115*g_deg2Rad, 0.607, 0.0, 90.0*g_deg2Rad, 0.0,
		 -65*g_deg2Rad, 0.607, 0.0, 90.0*g_deg2Rad, 0.0,
 		 -40*g_deg2Rad, 0.779, 0.0, 90.0*g_deg2Rad, 0.0];
	

END_VAR

// ---- GVLs/SlaveArms/GVL_SlaveControlParameters.TcGVL
{attribute 'global_init_slot' := '49991'}
VAR_GLOBAL CONSTANT
	// slave arm joint position controller parameters
	g_posKp :ARRAY[1..g_sJntNum] OF LREAL :=[2000.0, 2000.0, 18000.0, 5(5)];
	g_posKd :ARRAY[1..g_sJntNum] OF LREAL :=[200.0, 200.0, 200.0,5(0.25)];
	g_posKi :ARRAY[1..g_sJntNum] OF LREAL :=[20000.0, 20000.0, 30000.0, 5(10.0)];
	g_posKiLimit :ARRAY[1..g_sJntNum] OF LREAL :=[2500,2500,  250, 5(75)];// define in current
	g_posCtrlLimit :ARRAY[1..g_sJntNum] OF LREAL :=[5600,5600,  500, 5(250)];// define in current
	
	// control tolerance
	g_jntCtrlAngTolLow :LREAL :=0.2*g_deg2Rad;
	g_jntCtrlAngTolHigh :LREAL :=1*g_deg2Rad;
	g_cartCtrlPosTolLow :LREAL :=0.0002;
	g_cartCtrlOriTolLow :LREAL :=0.2*g_deg2Rad;
	g_cartCtrlPosTolHigh :LREAL :=0.001;
	g_cartCtrlOriTolHigh :LREAL :=1*g_deg2Rad;
	
	// filter cut-off frequency for velocity and torque
	g_curJntVelLpfCutoffFreq :LREAL := 30;
	g_cmdJntTrqLpfCutoffFreq :LREAL := 300;
	g_curJntTrqLpfCutoffFreq :LREAL := 300;
		
	// controller would keep command unchanged when error 
	// between command and current value is less than this value
	g_jntCtrlErrForCmdHold :LREAL :=1.0*g_deg2Rad;
	
	// joint is assumed to be static if velocity is less than this value
	g_jntStaticVelThres :LREAL :=0.2*g_deg2Rad;
	
	// joint velocity threshold for full friction compensation
	g_fullFrictionVel :LREAL :=2.0*g_deg2Rad;
	
	// friciton compensation scael
	g_frictionCompScale :LREAL := 0.8;
	
END_VAR

// ---- GVLs/SlaveArms/GVL_SlaveJointEncoderCaliData.TcGVL
{attribute 'qualified_only'}
// Robot4 --joints parameters of slave arms
VAR_GLOBAL CONSTANT
	// absolute encoder value at minimal joint positon
	g_minLinkEncoder :ARRAY[1..g_sArmNum, 1..g_sJntNum] OF DINT :=
		[5070618, 12248428, 9957376, 0, 0, 0, 0, 0,
		 4919708, 12165470, 13694272, 0, 0, 0, 0, 0,
		 9158200, 3936684, 16444112, 0, 0, 0, 0, 0,
		 13295020, 16357370, 9921792, 0, 0, 0, 0, 0];
		 
	// absolute encoder value at maximum joint positon
	g_maxLinkEncoder :ARRAY[1..g_sArmNum, 1..g_sJntNum] OF DINT :=
		[2939662, 5069530, 2375904, 0, 0, 0, 0, 0,
		2804134, 4974626, 6119888, 0, 0, 0, 0, 0,
		 6996994, 13526094, 8890176, 0, 0, 0, 0, 0,
		 11165812, 9145900, 2372960, 0, 0, 0, 0, 0];
	
	// absolute encoder value at calibrated positon
	g_caliLinkEncoder :ARRAY[1..g_sArmNum, 1..g_sJntNum] OF DINT :=
		[12427638, 8080000, 2375904, 15243664, 15283488, 7042832, 6950144, 7012272,
		12242476, 7980988, 6119888, 15217500, 15280288, 6866960, 6936528, 6826016,
		 16513242, 16579922, 8890176, 15265256, 15406944, 6400940, 6866960, 6902000,
		 3889656, 12177274, 2372960,15290800, 15066000, 6861290, 6710544, 6927488];
	
	 // if absolute encoder value cross zeros within joint motion range
	 // NOTICE: joint 7 is always 0.
	g_linkEncZeroCross :ARRAY[1..g_sArmNum, 1..g_sJntNum] OF INT :=
		[1, 0, 1, 1, 1, 1, 1, 1,
		 1, 0, 1, 1, 1, 1, 1, 1,
		 1, 1, 1, 1, 1, 1, 1, 1,
		 1, 0, 1, 1, 1, 1, 1, 1];
		 
	 // joint SDO address
	g_slaveArmNetID: ARRAY[1..4] OF T_AmsNetId:=['169.254.186.39.3.1','169.254.186.39.8.1','169.254.186.39.9.1','169.254.186.39.10.1'];
	g_slaveJointNetPort:ARRAY[1..g_sArmNum,1..g_sJntNum] OF UINT :=[
		1006,	1007,	1008,	2(1009),	3(1010),
		1006,	1007,	1008,	2(1009),	3(1010),
		1006,	1007,	1008,	2(1009),	3(1010),
		1006,	1007,	1008,	2(1009),	3(1010)];
		
//################ DO NOT modify parameters below ###########################
	// abolute encoder expanded limit buffer in case there is calibrtion error at limit position
	g_linkEncLimitBuffer : DINT := 100000;
	
	// absolute encoder direction
	g_asbEncoderDir :ARRAY[1..g_sJntNum] OF INT :=[1, -1, 1, 1, 1, 1, 1, 1];
	
	// flag if joint can rotate multiple cycles
	g_multipleCyclesJoint :ARRAY[1..g_sArmNum, 1..g_sJntNum] OF INT :=
		[0, 0, 0, 1, 1, 1, 1, 1,
		 0, 0, 0, 1, 1, 1, 1, 1,
		 0, 0, 0, 1, 1, 1, 1, 1,
		 0, 0, 0, 1, 1, 1, 1, 1];
		 
	// joint position at link encoder calibrated point
	g_linkEncCaliJntPos :ARRAY[1..g_sJntNum] OF LREAL :=
		[0.0, -PI/2, 0.581633, 5(0.0)];

	
END_VAR

// ---- FBs_CartControlles/I_CartJointCtrl.TcIO
INTERFACE I_CartJointCtrl

METHOD init : BOOL
VAR_IN_OUT CONSTANT
	i_slaveCart	:FB_SlaveCart;
END_VAR
VAR_IN_OUT 
	r_cartCtrlCmd :ST_SlaveArmCtrlCmds;
END_VAR
END_METHOD

PROPERTY isFinished : BOOL
GET
END_GET
END_PROPERTY

METHOD reset : BOOL
VAR_INPUT
END_VAR
END_METHOD

METHOD run : BOOL
VAR_IN_OUT CONSTANT
	i_slaveCart	:FB_SlaveCart;
END_VAR
VAR_IN_OUT 
	r_cartCtrlCmd :ST_SlaveArmCtrlCmds;
END_VAR
END_METHOD

END_INTERFACE

// ---- FBs_Auxiliary/FB_setupAdjustDetect.TcPOU
FUNCTION_BLOCK FB_setupAdjustDetect
VAR_INPUT
END_VAR
VAR_OUTPUT
END_VAR
VAR
	m_manualAdjustOnCounts :INT :=0;
	m_adjustOnCountThres :INT :=50;
END_VAR

METHOD run : BOOL
VAR_INPUT
	IOValue :UDINT;
END_VAR

VAR_OUTPUT
	
END_VAR
// manuel adjust io is 5th bit 
IF 16=(IOValue AND 10#16) THEN
	m_manualAdjustOnCounts :=MIN(m_manualAdjustOnCounts +1,m_adjustOnCountThres);
ELSE
	m_manualAdjustOnCounts :=0;
END_IF

run := m_manualAdjustOnCounts >= m_adjustOnCountThres;
END_METHOD

END_FUNCTION_BLOCK

// ---- FBs_Auxiliary/FB_TrocarDetect.TcPOU
FUNCTION_BLOCK FB_TrocarDetect
VAR_INPUT
END_VAR
VAR_OUTPUT
END_VAR
VAR
	m_trocarOnCounts :INT :=0;
	m_trocarOnCountThres :INT :=50;
END_VAR

// check if instrument is on
METHOD run : BOOL
VAR_INPUT
	IOValue :UDINT;
END_VAR
// trocar io is 5th bit 
IF 32=(IOValue AND 10#32) THEN
	m_trocarOnCounts :=MIN(m_trocarOnCounts +1,m_trocarOnCountThres);
ELSE
	m_trocarOnCounts :=0;
END_IF

run := m_trocarOnCounts >= m_trocarOnCountThres;
END_METHOD

END_FUNCTION_BLOCK

// ---- FBs_Auxiliary/FB_PanelDetect.TcPOU
FUNCTION_BLOCK FB_PanelDetect
VAR_INPUT
END_VAR
VAR_OUTPUT
END_VAR
VAR
	m_panelOnCounts :INT :=0;
	m_panelOnCountThres :INT :=50;
END_VAR

// check if panel is on
METHOD run : BOOL
VAR_INPUT
	IOValue :UDINT;
END_VAR
//Panel single  At installation--2#0000   not installation --2#0101
IF (IOValue AND 16#05) = 0 THEN
	m_panelOnCounts := MIN( m_panelOnCounts +1,m_panelOnCountThres);
ELSIF (IOValue AND 16#05) = 5  THEN
	m_panelOnCounts :=0;
END_IF
run := m_panelOnCounts >= m_panelOnCountThres;
END_METHOD

END_FUNCTION_BLOCK

// ---- FBs_Auxiliary/FB_InstrumentDetect.TcPOU
FUNCTION_BLOCK FB_InstrumentDetect
VAR_INPUT
END_VAR
VAR_OUTPUT
END_VAR
VAR
	m_instruOnCounts :INT :=0;
	m_InstruOnCountThres :INT :=50;
END_VAR

// check if instrument is on
METHOD run : BOOL
VAR_INPUT
	IOValue :UDINT;
END_VAR
//Instrument single   At installation--2#0*0*   not installation --2#1*1*  And Hall single --2#100 0000
IF (IOValue AND 16#A) = 0  THEN
	m_instruOnCounts := MIN( m_instruOnCounts +1,m_InstruOnCountThres);
ELSIF (IOValue AND 16#4A) = 10  THEN
	m_instruOnCounts :=0;
END_IF
run := m_instruOnCounts >= m_InstruOnCountThres;
END_METHOD

END_FUNCTION_BLOCK

// ---- FBs_CartControlles/FB_CartCtrlAsepticDeploy.TcPOU
FUNCTION_BLOCK FB_CartCtrlAsepticDeploy EXTENDS FB_CartCtrlBase
VAR_INPUT
END_VAR
VAR_OUTPUT
END_VAR
VAR

	m_actJntPos: Vec8d;
	m_tarJntPos: Vec8d;
	m_jntPosArrival : Vec8b;
	m_initActJntPos: Vec8d;
	m_initTarJntPos : Vec8d;
	m_incTarJntPos : Vec8d;

	// time threshold to 5-8joint after it's enabled
	m_cartAdjustStartWaitTime :LREAL := 0.2;
	
	//adjust start  time 
	m_adjustStartTime :LREAL;
	
	m_jntOTG :ARRAY[1..8] OF FB_secOrdTrajFilter;
	//m_trajPlan :ARRAY[1..8] OF TrapezoIDal_velocity_trajectory;
END_VAR

// override this function in each exact controller
METHOD PROTECTED calcCmdJntPos : BOOL
VAR_IN_OUT CONSTANT
	// slave cart joint data
	i_slaveCart :FB_SlaveCart;
END_VAR

VAR
	i:INT;
END_VAR
//In this method, 5 represents the pillar postion , 6 represents the beam rotation angle ,7 represents the beam stretch position ,8 represents the overhang angle
m_adjustStartTime :=LIMIT(0, m_adjustStartTime + g_cartCtrlCycleTime, 1);
m_actJntPos := i_slaveCart.curJntPos;
IF i_slaveCart.ctrlEnable.docking_enable THEN
	m_initTarJntPos := i_slaveCart.m_cartDataFromUI.m_cartSpecificPosDocking;
ELSIF i_slaveCart.ctrlEnable.draping_enable THEN
	m_initTarJntPos := i_slaveCart.m_cartDataFromUI.m_cartSpecificPosDraping;
END_IF

IF m_adjustStartTime >= m_cartAdjustStartWaitTime THEN
	FOR i := 5 TO 8 BY 1 DO
		IF ABS(m_initTarJntPos[i] - m_actJntPos[i]) <= GVL_CartControlParameters.g_jntCtrlAngTolHigh*2  THEN
			m_jntPosArrival[i] := TRUE;
		END_IF
		
		IF ABS(m_initTarJntPos[i] - m_tarJntPos[i]) <= GVL_CartControlParameters.g_jntCtrlAngTolHigh  THEN
			m_jntPosArrival[i-4] := TRUE;
		END_IF
		
		IF m_jntPosArrival[i-4] = FALSE THEN
			m_incTarJntPos[i] := m_incTarJntPos[i] + sign(m_initTarJntPos[i] - m_actJntPos[i]) * GVL_CartControlParameters.g_maxJntVel[i]/2 * g_cartCtrlCycleTime;
			m_tarJntPos[i] := m_actJntPos[i] + m_incTarJntPos[i];
		END_IF
	END_FOR
	
	IF m_jntPosArrival[5] AND m_jntPosArrival[6] AND m_jntPosArrival[7] AND m_jntPosArrival[8] THEN
		m_isFinished := TRUE;
	END_IF
	
	FOR i := 5 TO 8 BY 1 DO
		m_jntOTG[i].run(i_targetPos:= m_tarJntPos[i], i_targetVel:= 0.0, o_cmdAcc=> , o_cmdVel=> , o_cmdPos=>m_cmdJntPos[i] );
	END_FOR
END_IF
END_METHOD

// override this function in each exact controller
// NOTICE: set joint control mode here, and do some initialization if needed
METHOD PUBLIC init : BOOL
VAR_IN_OUT CONSTANT
	i_slaveCart	:FB_SlaveCart;
END_VAR
VAR_IN_OUT 
	r_cartCtrlCmd :ST_SlaveArmCtrlCmds;
END_VAR
VAR
	i : INT;
END_VAR
SUPER^.init(i_slaveCart,r_cartCtrlCmd);

m_jntEnableFlag[5] :=1;
m_jntEnableFlag[6] :=1;
m_jntEnableFlag[7] :=1;
m_jntEnableFlag[8] :=1;

m_jntOPMode[5]:= DriverOPMode_cspMZ;
m_jntOPMode[6]:= DriverOPMode_Pos;
m_jntOPMode[7]:= DriverOPMode_Pos;
m_jntOPMode[8]:= DriverOPMode_Pos;

m_initActJntPos:=i_slaveCart.curJntPos;
m_jntPosArrival := g_zeroVec8b;
m_incTarJntPos := g_zeroVec8d;
m_tarJntPos := g_zeroVec8d;
m_jntPosArrival := g_zeroVec8b;

IF i_slaveCart.ctrlEnable.docking_enable THEN
	m_initTarJntPos := i_slaveCart.m_cartDataFromUI.m_cartSpecificPosDocking;
ELSIF i_slaveCart.ctrlEnable.draping_enable THEN
	m_initTarJntPos := i_slaveCart.m_cartDataFromUI.m_cartSpecificPosDraping;
END_IF

FOR i := 1 TO 4 BY 1 DO
	m_jntOTG[i+4].init(i_curCmdPos:= m_cmdJntPos[i+4], i_curCmdVel:= 0, i_maxV:=GVL_CartControlParameters.g_maxJntVel[i+4]/2 , i_maxA:=GVL_CartControlParameters.g_maxJntAcc[i+4]/2 , i_Ts:=g_cartCtrlCycleTime );
END_FOR
//m_initTarJntPos := m_tarJntPos;
m_adjustStartTime := 0;
// update commands to arm
copyCmds(r_cartCtrlCmd);
END_METHOD

END_FUNCTION_BLOCK

// ---- FBs_CartControlles/FB_CartCtrlBase.TcPOU
// Slave Arm Base Controller, Hold at Current Posture
FUNCTION_BLOCK FB_CartCtrlBase IMPLEMENTS I_CartJointCtrl
VAR_INPUT
END_VAR
VAR_OUTPUT
END_VAR
VAR
	// flag if the controller has finished all its jobs
	m_isFinished:BOOL:=FALSE;
	
	// controller execute time period
	m_timePeriod :LREAL:=0;
	
	// flag to hold last commands
	m_holdLastCmds :BOOL := FALSE;
	
	// arm control data
	// NOTE: simulated joint position is usd for kinematic controller 
	//		while command joint position is used for real robot controller
	// 		They are identical for the most time, but in some cases, simulated position is filted to get command one 
	m_cmdJntPos : VEC8d; 
	m_cmdJntVel : VEC8d;
	m_cmdJntAcc : VEC8d;
	m_cmdJntTrq : VEC8d;
	m_jntOPMode : Vec8i;
	m_jntEnableFlag :Vec8i;

	
END_VAR

// override this function in each exact controller
METHOD PROTECTED calcCmdJntPos : BOOL
VAR_IN_OUT CONSTANT
	// slave cart joint data
	i_slaveCart :FB_SlaveCart;
END_VAR
IF isFinished THEN
	RETURN;
END_IF
END_METHOD

// override this function in each exact controller
METHOD PROTECTED calcCmdJntVel : BOOL
VAR_IN_OUT CONSTANT
	// slave cart joint data
	i_slaveCart :FB_SlaveCart;
END_VAR
IF isFinished THEN
	RETURN;
END_IF

// set joint torque to zero in default
//m_cmdJntVel := g_zeroVec8d;
END_METHOD

METHOD checkToHoldLastCmds : BOOL
VAR_IN_OUT CONSTANT
	// slave cart joint data
	i_slaveCart :FB_SlaveCart;
END_VAR
VAR
	j:INT;
	maxJntErr:LREAL;
	jntCtrlErr:Vec7d;
END_VAR
// check if to hold the command joint position unchanged
vecSub(i_slaveCart.m_cmdJntPos, i_slaveCart.m_curJntPos,jntCtrlErr);
maxJntErr:=0.0;
FOR j:=1 TO g_sJntNum DO
	maxJntErr:= MAX(maxJntErr, ABS(jntCtrlErr[j]));
END_FOR

checkToHoldLastCmds := (maxJntErr<GVL_SlaveControlParameters.g_jntCtrlErrForCmdHold);
END_METHOD

METHOD copyCmds : BOOL
VAR_IN_OUT 
	r_cartCtrlCmd :ST_SlaveArmCtrlCmds;
END_VAR
r_cartCtrlCmd.m_jntEnableFlag :=m_jntEnableFlag;
r_cartCtrlCmd.m_cmdJntPos:=m_cmdJntPos;
r_cartCtrlCmd.m_cmdJntVel:=m_cmdJntVel;
r_cartCtrlCmd.m_cmdJntAcc:=m_cmdJntAcc;
r_cartCtrlCmd.m_cmdJntTrq:=m_cmdJntTrq;
r_cartCtrlCmd.m_jntOPMode:=m_jntOPMode;
END_METHOD

// override this function in each exact controller
// NOTICE: set joint control mode here, and do some initialization if needed
METHOD PUBLIC init : BOOL
VAR_IN_OUT CONSTANT
	// slave cart joint data
	i_slaveCart :FB_SlaveCart;
END_VAR
VAR_IN_OUT 
	r_cartCtrlCmd :ST_SlaveArmCtrlCmds;
END_VAR
m_timePeriod:=0;
m_jntEnableFlag :=g_zeroVec8i;
m_jntOPMode:=g_slaveAllPosMode;

IF FALSE = m_holdLastCmds THEN
	m_cmdJntPos:=i_slaveCart.m_curJntPos;
ELSE
	m_cmdJntPos:=r_cartCtrlCmd.m_cmdJntPos;
END_IF

m_cmdJntVel:=g_zeroVec8d;
m_cmdJntAcc:=g_zeroVec8d;
m_cmdJntTrq:=g_zeroVec8d;

// update commands to arm
copyCmds(r_cartCtrlCmd);
END_METHOD

PROPERTY isFinished : BOOL
GET
isFinished:=m_isFinished;
END_GET
END_PROPERTY

{warning '添加方法实现'}
METHOD reset : BOOL
m_isFinished:=FALSE;
m_timePeriod:=0;
END_METHOD

{warning '添加方法实现'}
METHOD run : BOOL
VAR_IN_OUT CONSTANT
	// slave cart joint data
	i_slaveCart :FB_SlaveCart;
END_VAR
VAR_IN_OUT
	r_cartCtrlCmd :ST_SlaveArmCtrlCmds;
END_VAR
VAR
	i:INT;
END_VAR
IF m_isFinished THEN
	RETURN;
END_IF

// check if arm enabled
//IF FALSE = i_slaveCartJoint.isEnabled(m_jntEnableFlag) THEN
//	RETURN;
//END_IF

// calculate command joint position--Motion control
calcCmdJntPos( i_slaveCart);

// calculate command joint torque -- Force control
calcCmdJntVel(i_slaveCart);

// update commands to arm
copyCmds(r_cartCtrlCmd);

// update time period
m_timePeriod := m_timePeriod+g_slaveArmCtrlCycleTime;
END_METHOD

END_FUNCTION_BLOCK

// ---- FBs_CartControlles/FB_CartCtrlError.TcPOU
FUNCTION_BLOCK FB_CartCtrlError EXTENDS FB_CartCtrlBase
VAR_INPUT
END_VAR
VAR_OUTPUT
END_VAR
VAR
END_VAR

// override this function in each exact controller
METHOD PROTECTED calcCmdJntPos : BOOL
VAR_IN_OUT CONSTANT
	// slave cart joint data
	i_slaveCart :FB_SlaveCart;
END_VAR
m_cmdJntPos := i_slaveCart.curJntPos;
END_METHOD

// override this function in each exact controller
// NOTICE: set joint control mode here, and do some initialization if needed
METHOD PUBLIC init : BOOL
VAR_IN_OUT CONSTANT
	i_slaveCart	:FB_SlaveCart;
END_VAR
VAR_IN_OUT 
	r_cartCtrlCmd :ST_SlaveArmCtrlCmds;
END_VAR
SUPER^.init(i_slaveCart,r_cartCtrlCmd);

// update commands to arm
copyCmds(r_cartCtrlCmd);
END_METHOD

END_FUNCTION_BLOCK

// ---- FBs_CartControlles/FB_CartCtrlReady.TcPOU
FUNCTION_BLOCK FB_CartCtrlReady EXTENDS FB_CartCtrlBase
VAR_INPUT
END_VAR
VAR_OUTPUT
END_VAR
VAR
END_VAR

// override this function in each exact controller
METHOD PROTECTED calcCmdJntPos : BOOL
VAR_IN_OUT CONSTANT
	// slave cart joint data
	i_slaveCart :FB_SlaveCart;
END_VAR
m_cmdJntPos := i_slaveCart.curJntPos;
END_METHOD

// override this function in each exact controller
// NOTICE: set joint control mode here, and do some initialization if needed
METHOD PUBLIC init : BOOL
VAR_IN_OUT CONSTANT
	i_slaveCart	:FB_SlaveCart;
END_VAR
VAR_IN_OUT 
	r_cartCtrlCmd :ST_SlaveArmCtrlCmds;
END_VAR
SUPER^.init(i_slaveCart,r_cartCtrlCmd);

// update commands to arm
copyCmds(r_cartCtrlCmd);
END_METHOD

END_FUNCTION_BLOCK

// ---- FBs_CartControlles/FB_CartCtrlRotaOverhang.TcPOU
FUNCTION_BLOCK FB_CartCtrlRotaOverhang EXTENDS FB_CartCtrlBase
VAR_INPUT
END_VAR
VAR_OUTPUT
END_VAR
VAR

	m_actJntPos: Vec8d;
	m_tarJntPos: Vec8d;
	m_cmdJntDir : INT;
	m_rotaAngle:LREAL:=2.5 * g_deg2Rad ;
	m_initJntPos : LREAL;
	m_tarJntInc : LREAL;

	m_carJntSoftwareLimit :ARRAY [5..8] OF LREAL := [0.005, 2*g_deg2Rad, 0.005, 2*g_deg2Rad];
	
	// time threshold to 5-8joint after it's enabled
	m_cartAdjustStartWaitTime :LREAL := 0.2;
	
	//adjust start  time 
	m_adjustStartTime :LREAL;

	m_jntOTG : FB_secOrdTrajFilter;
END_VAR

// override this function in each exact controller
METHOD PROTECTED calcCmdJntPos : BOOL
VAR_IN_OUT CONSTANT
	// slave cart joint data
	i_slaveCart :FB_SlaveCart;
END_VAR

VAR
	i:INT;
END_VAR
//In this method, 8 represents the overhang angle
m_adjustStartTime :=LIMIT(0, m_adjustStartTime + g_cartCtrlCycleTime, 1);
m_actJntPos := i_slaveCart.curJntPos;
IF i_slaveCart.m_rotaOverhangOnFlag = 1 THEN
	m_cmdJntDir := -1;
ELSIF i_slaveCart.m_rotaOverhangOnFlag = 2 THEN
	m_cmdJntDir := 1;
END_IF

IF m_adjustStartTime > m_cartAdjustStartWaitTime THEN
	m_tarJntInc := m_tarJntInc + m_cmdJntDir * m_rotaAngle * g_cartCtrlCycleTime;
	
	m_tarJntPos[8] := LIMIT(GVL_CartMotorParameters.g_minJntPos[8] + m_carJntSoftwareLimit[8], m_initJntPos + m_tarJntInc, GVL_CartMotorParameters.g_maxJntPos[8] - m_carJntSoftwareLimit[8]);

	m_jntOTG.run(i_targetPos:= m_tarJntPos[8], i_targetVel:= 0.0, o_cmdAcc=> , o_cmdVel=> , o_cmdPos=>m_cmdJntPos[8] );
END_IF
END_METHOD

// override this function in each exact controller
// NOTICE: set joint control mode here, and do some initialization if needed
METHOD PUBLIC init : BOOL
VAR_IN_OUT CONSTANT
	i_slaveCart	:FB_SlaveCart;
END_VAR
VAR_IN_OUT 
	r_cartCtrlCmd :ST_SlaveArmCtrlCmds;
END_VAR
VAR
	i:INT;
END_VAR
SUPER^.init(i_slaveCart,r_cartCtrlCmd);

m_jntEnableFlag[8] :=1;

m_jntOPMode[8]:= DriverOPMode_Pos;
m_initJntPos := i_slaveCart.curJntPos[8];
m_tarJntInc := 0;

m_jntOTG.init(i_curCmdPos:= m_cmdJntPos[8], i_curCmdVel:= 0, i_maxV:=GVL_CartControlParameters.g_maxJntVel[8] , i_maxA:=GVL_CartControlParameters.g_maxJntAcc[8] , i_Ts:=g_cartCtrlCycleTime );


m_adjustStartTime := 0;
// update commands to arm
copyCmds(r_cartCtrlCmd);
END_METHOD

END_FUNCTION_BLOCK

// ---- FBs_CartControlles/FB_CartCtrlSlowDown.TcPOU
FUNCTION_BLOCK FB_CartCtrlSlowDown EXTENDS FB_CartCtrlBase
VAR_INPUT
END_VAR
VAR_OUTPUT
END_VAR
VAR

	m_tarPosInc: Vec8d;
	m_trajVel : Vec8d;
	m_initVel : Vec8d;
	m_initPos : Vec8d;
	m_initDec : Vec8d;
	
	//slow down and stop time
	m_incSlowStopTime :LREAL;
	m_slowStopTime :LREAL :=0.5;
	
	// filter cut-off frequency for cart drive force 
	m_cmdJoystickLpfCutoffFreq : LREAL :=8;
	m_cartCtrlFreq :LREAL:=8000;
END_VAR

// override this function in each exact controller
METHOD PROTECTED calcCmdJntPos : BOOL
VAR_IN_OUT CONSTANT
	// slave cart joint data
	i_slaveCart :FB_SlaveCart;
END_VAR

VAR
	i:INT;
END_VAR
//In this method, 5 represents the pillar postion , 6 represents the beam rotation angle ,7 represents the beam stretch position ,8 represents the overhang angle
m_incSlowStopTime :=LIMIT(0, m_incSlowStopTime + g_cartCtrlCycleTime, 1);

FOR i := 1 TO 8 BY 1 DO
	m_trajVel[i] := m_initVel[i] - m_initDec[i] * m_incSlowStopTime;
	IF ABS(m_initVel[i]) < ABS(m_initDec[i]) * m_incSlowStopTime THEN
		m_trajVel[i]:=0;
	END_IF
	m_tarPosInc[i] := m_tarPosInc[i] + m_trajVel[i] * g_cartCtrlCycleTime;
	m_cmdJntPos[i] := m_initPos[i] + m_tarPosInc[i];
END_FOR

IF m_incSlowStopTime >= m_slowStopTime THEN//m_slowStopTime THEN
	m_isFinished := TRUE;
END_IF
END_METHOD

// override this function in each exact controller
// NOTICE: set joint control mode here, and do some initialization if needed
METHOD PUBLIC init : BOOL
VAR_IN_OUT CONSTANT
	i_slaveCart	:FB_SlaveCart;
END_VAR
VAR_IN_OUT 
	r_cartCtrlCmd :ST_SlaveArmCtrlCmds;
END_VAR

m_cmdJntPos:=r_cartCtrlCmd.m_cmdJntPos;
m_initPos := m_cmdJntPos;

m_jntEnableFlag :=r_cartCtrlCmd.m_jntEnableFlag;

m_jntOPMode[5]:= DriverOPMode_cspMZ;
m_jntOPMode[6]:= DriverOPMode_Pos;
m_jntOPMode[7]:= DriverOPMode_Pos;
m_jntOPMode[8]:= DriverOPMode_Pos;

m_trajVel[5] := 0;
m_trajVel[6] := 0;
m_trajVel[7] := 0;
m_trajVel[8] := 0;

m_tarPosInc[5] := 0;
m_tarPosInc[6] := 0;
m_tarPosInc[7] := 0;
m_tarPosInc[8] := 0;


m_incSlowStopTime := 0;

m_initVel[5] := LIMIT(-GVL_CartMotorParameters.g_maxJntVel[5], i_slaveCart.curJntVel[5], GVL_CartMotorParameters.g_maxJntVel[5]);
m_initVel[6] := LIMIT(-GVL_CartMotorParameters.g_maxJntVel[6], i_slaveCart.curJntVel[6], GVL_CartMotorParameters.g_maxJntVel[6]);
m_initVel[7] := LIMIT(-GVL_CartMotorParameters.g_maxJntVel[7], i_slaveCart.curJntVel[7], GVL_CartMotorParameters.g_maxJntVel[7]);
m_initVel[8] := LIMIT(-GVL_CartMotorParameters.g_maxJntVel[8], i_slaveCart.curJntVel[8], GVL_CartMotorParameters.g_maxJntVel[8]);


m_initDec[5] := sign(m_initVel[5])*GVL_CartMotorParameters.g_maxJntVel[5];
m_initDec[6] := sign(m_initVel[6])*GVL_CartMotorParameters.g_maxJntVel[6];
m_initDec[7] := sign(m_initVel[7])*GVL_CartMotorParameters.g_maxJntVel[7];
m_initDec[8] := sign(m_initVel[8])*GVL_CartMotorParameters.g_maxJntVel[8];


m_slowStopTime := 0.5;
// update commands to arm
copyCmds(r_cartCtrlCmd);
END_METHOD

END_FUNCTION_BLOCK

// ---- FBs_RobotDynamics/FB_SlaveGravity.TcPOU
FUNCTION_BLOCK FB_SlaveGravity
VAR_INPUT
END_VAR
VAR
	m_armIdx :INT ;

	// current arm parameters
	m_armParams :ARRAY[1..5] OF LREAL;

END_VAR

METHOD getRegMat : BOOL
VAR_INPUT
	// joint position of setup joint, joint6-8
	setupAng :LREAL;
	q1: LREAL;
	q2: LREAL;
	q3: LREAL;
END_VAR

VAR
	s0,c0, s1,c1,s2, c2,d3 :LREAL;
END_VAR

VAR_OUTPUT
	o_regMat:ARRAY[1..3,1..5] OF LREAL;
END_VAR
s0:=SIN(setupAng);
c0:=COS(setupAng);
s1:=SIN(q1);
c1:=COS(q1);
s2:=SIN(q2);
c2:=COS(q2);
d3:=q3;

// joint1
o_regMat[1,1] :=s0*s1*s2*d3;
o_regMat[1,2] :=  s0*s1;
o_regMat[1,3] := -s0*c1;
o_regMat[1,4] := s0*s1*s2;
o_regMat[1,5] := s0*c2*s1 ;

// joint2 
o_regMat[2,1] :=  - (c0*s2*d3+s0*c1*c2*d3);
o_regMat[2,2] := 0;
o_regMat[2,3] := 0;
o_regMat[2,4] :=  - (c0*s2+s0*c1*c2);
o_regMat[2,5] := s0*c1*s2- c0*c2;

// joint3
o_regMat[3,1] :=c0*c2 - s0*c1*s2;
o_regMat[3,2] :=0;
o_regMat[3,3] :=0;
o_regMat[3,4] :=0;
o_regMat[3,5] :=0;
END_METHOD

METHOD init : BOOL
VAR_INPUT
	i_armIdx :INT;
END_VAR
m_armIdx :=i_armIdx;
END_METHOD

METHOD run : Vec3d
VAR_IN_OUT CONSTANT
	// setup joint5 angle
	i_setupPos :LREAL;
	
	// slave joint angle
	i_slaveJntPos :Vec8d;
	
	// instrument
	i_instruStatus :ST_InstruStatus;
END_VAR
VAR
	q1, q2, q3 :LREAL;
	i,j:INT;
	
	// gravity regression matrix
	regMat:ARRAY[1..3,1..5] OF LREAL;
END_VAR
q1 := i_slaveJntPos[1];
q2 := i_slaveJntPos[2];
q3 := i_slaveJntPos[3];


// get regression matrx
getRegMat(i_setupPos, q1, q2, q3, o_regMat=>regMat);

// determine current arm parameters
IF FALSE = i_instruStatus.m_ready THEN
	// arm only
	FOR i:=1 TO 5 DO
		m_armParams[i]:=GVL_SlaveArmDynamics.g_gravityParam[m_armIdx,i];
	END_FOR

// endoscope
ELSIF InstruType_endoscope = i_instruStatus.m_type THEN 
	FOR i:=1 TO 5 DO
		m_armParams[i]:=GVL_SlaveArmDynamics.g_gravityParam[m_armIdx,i]+GVL_SlaveArmDynamics.g_gravityEndoscope[i];
	END_FOR

// instrument
ELSE
	FOR i:=1 TO 5 DO
		m_armParams[i]:=GVL_SlaveArmDynamics.g_gravityParam[m_armIdx,i]+GVL_SlaveArmDynamics.g_gravityInstrument[i];
	END_FOR
// TODO:Trocar
END_IF

// calculate gravity torque
FOR i:=1 TO 3 DO
	run[i]:=0;
	FOR j:=1 TO 5 DO
		run[i]:=run[i]+regMat[i,j]*m_armParams[j];
	END_FOR
END_FOR
END_METHOD

END_FUNCTION_BLOCK

// ---- FBs_RobotDynamics/FB_SetupGravity.TcPOU
FUNCTION_BLOCK FB_SetupGravity
VAR_INPUT
END_VAR
VAR
	m_armIdx :INT ;

	// current arm parameters
	m_armParams :ARRAY[1..7] OF LREAL;

	// gravity regression matrix
	regMat:ARRAY[1..7] OF LREAL;
	
	m_graivty :LREAL;
END_VAR

METHOD getRegMat : BOOL
VAR_INPUT
	// joint position of setup joint, joint6-8
	setupAng :LREAL;
	q1: LREAL;
	q2: LREAL;
	q3: LREAL;
END_VAR

VAR
	s0,c0,s1,c1,s2, c2,d3 :LREAL;
END_VAR

VAR_OUTPUT
	o_regMat:ARRAY[1..7] OF LREAL;
END_VAR
s0:= SIN(setUpAng);
c0:= COS(setUpAng);
s1:=SIN(q1);
c1:=COS(q1);
s2:=SIN(q2);
c2:=COS(q2);
d3:=q3;

// setup joint
o_regMat[1] :=c0;
o_regMat[2] := s0;
o_regMat[3] :=-(c2*s0*d3+c0*c1*s2*d3);
o_regMat[4] :=  -c0*c1;
o_regMat[5] :=  -c0*s1;
o_regMat[6] := - (c0*c1*s2+c2*s0);
o_regMat[7] :=  s0*s2- c0*c1*c2  ;
END_METHOD

METHOD init : BOOL
VAR_INPUT
	i_armIdx :INT;
END_VAR
m_armIdx :=i_armIdx;
END_METHOD

METHOD run : BOOL
VAR_IN_OUT CONSTANT
	// setup joint angle
	i_setupJntPos :Vec5d;
	
	// slave joint angle
	i_slaveJntPos :Vec8d;
	
	// instrument
	i_instruStatus :ST_InstruStatus;
END_VAR
VAR_OUTPUT
	// setup joint3 gravity
	o_jnt3Gravity :LREAL;
	
	// setup joint5 gravity
	o_jnt5Gravity :LREAL;
END_VAR
VAR
	setupPos, q1, q2, q3 :LREAL;
	i,j:INT;
	
	gravityTrq :Vec4d;

END_VAR
setupPos:=i_setupJntPos[5];
q1 := i_slaveJntPos[1];
q2 := i_slaveJntPos[2];
q3 := i_slaveJntPos[3];

// get regression matrx
getRegMat(setupPos, q1, q2, q3, o_regMat=>regMat);

// determine current arm parameters
m_armParams[1] := GVL_SetupArmDynamics.g_setupJnt5GravityParam[m_armIdx,1];
m_armParams[2] := GVL_SetupArmDynamics.g_setupJnt5GravityParam[m_armIdx,2];
IF FALSE = i_instruStatus.m_ready THEN
	// arm only
	FOR i:=1 TO 5 DO
		m_armParams[i+2]:= GVL_SlaveArmDynamics.g_gravityParam[m_armIdx,i];
	END_FOR

// endoscope
ELSIF InstruType_endoscope = i_instruStatus.m_type THEN 
	FOR i:=1 TO 5 DO
		m_armParams[i+2]:=GVL_SlaveArmDynamics.g_gravityParam[m_armIdx,i]+GVL_SlaveArmDynamics.g_gravityEndoscope[i];
	END_FOR

// instrument
ELSE
	FOR i:=1 TO 5 DO
		m_armParams[i+2]:=GVL_SlaveArmDynamics.g_gravityParam[m_armIdx,i]+GVL_SlaveArmDynamics.g_gravityInstrument[i];
	END_FOR
// TODO:Trocar
END_IF

// calculate gravity torque
o_jnt5Gravity:=0;
FOR j:=1 TO 7 DO
	o_jnt5Gravity:=o_jnt5Gravity+regMat[j]*m_armParams[j];
END_FOR
m_graivty := o_jnt5Gravity;

o_jnt3Gravity:= setupJnt3Gravity(i_setupJntPos[3]);
END_METHOD

METHOD setupJnt3Gravity : LREAL
VAR_INPUT
	i_jnt3Pos :LREAL;
END_VAR
VAR
	q:LREAL;
END_VAR
q := LIMIT(GVL_SetupArmDynamics.g_setupJnt3GravityPosRange[m_armIdx,1], i_jnt3Pos, GVL_SetupArmDynamics.g_setupJnt3GravityPosRange[m_armIdx,2]);
setupJnt3Gravity:=GVL_SetupArmDynamics.g_setupJnt3GravityParams[m_armIdx,1]*EXPT(q,3)+GVL_SetupArmDynamics.g_setupJnt3GravityParams[m_armIdx,2]*EXPT(q,2)+
				GVL_SetupArmDynamics.g_setupJnt3GravityParams[m_armIdx,3]*q+GVL_SetupArmDynamics.g_setupJnt3GravityParams[m_armIdx,4];
END_METHOD

END_FUNCTION_BLOCK

// ---- FBs_Robots/FB_CartRobot.TcPOU
FUNCTION_BLOCK FB_CartRobot
VAR_INPUT
END_VAR
VAR_OUTPUT
END_VAR
VAR

	m_slaveCart: FB_SlaveCart;		
	
	// input arm button 
	m_carHandChassisDriveUnlock AT%I* :ARRAY [1..2] OF BOOL;

	m_joystickData:Vec8d;

	//m_cartDrapingState : UINT;
	//m_cartDockingState : UINT;
	// all cart controller instance 
	m_cartCtrlFactory :ARRAY[1..CartJointState_totalNum] OF I_CartJointCtrl;
	
	m_cartState:E_CartJointState:=CartJointState_Init;
	m_lastCartState:E_CartJointState:=CartJointState_Init;
	m_nextCartState:E_CartJointState:=CartJointState_Init;
	
	// flag if cart joint self-check passed
	m_selfCheckPass:  BOOL :=FALSE;
	
	// all cart controller instance 
	m_cartError :FB_CartCtrlError;
	m_cartInit :FB_CartCtrlInit;
	m_cartReady :FB_CartCtrlReady;
	m_cartInSurgery :FB_CartCtrlInSurgery;
	m_cartMotionCar :FB_CartCtrlMotionCar;
	m_cartAsepticDeploy :FB_CartCtrlAsepticDeploy;
	m_cartAdjust :FB_CartCtrlAdjust;
	m_cartRotaOverhang :FB_CartCtrlRotaOverhang;
	m_cartSlowStop : FB_CartCtrlSlowDown;
	
	// cart controller interface
	m_cartCtrl : I_CartJointCtrl;
	m_cartCtrlCmds : ST_SlaveArmCtrlCmds;
	
END_VAR

METHOD getStatus : BOOL
VAR_IN_OUT
	
	r_cartStatus :ST_CartStatus;	

	// cart joint data
	r_cartJointsData :ST_CartJointData;
END_VAR

//r_cartStatus.m_CartState:=m_cartState;
END_METHOD

METHOD init : BOOL
VAR_INPUT
END_VAR
VAR
	i:INT;
END_VAR

m_slaveCart.init();
m_cartState := CartJointState_Init;
m_lastCartState := CartJointState_Init;
m_nextCartState := CartJointState_Init;
m_selfCheckPass := FALSE;

//command init
m_cartCtrlCmds.m_jntEnableFlag := g_zeroVec8i;
m_cartCtrlCmds.m_jntOPMode := g_slaveAllPosMode;
m_cartCtrlCmds.m_cmdJntPos := m_slaveCart.m_curJntPos;
m_cartCtrlCmds.m_cmdJntVel := g_zeroVec8d;
m_cartCtrlCmds.m_cmdJntAcc := g_zeroVec8d;
m_cartCtrlCmds.m_cmdJntTrq := g_zeroVec8d;


// generate controller factory
//m_cartCtrlFactory[CartJointState_Error] := m_cartError;
m_cartCtrlFactory[CartJointState_Init] := m_cartInit;
m_cartCtrlFactory[CartJointState_Ready] := m_cartReady;
m_cartCtrlFactory[CartJointState_InSurgery] := m_cartInSurgery;
m_cartCtrlFactory[CartJointState_Movement] := m_cartMotionCar;
m_cartCtrlFactory[CartJointState_HangAdjust] := m_cartAdjust;
m_cartCtrlFactory[CartJointState_AsepticDeployment] := m_cartAsepticDeploy;
m_cartCtrlFactory[CartJointState_RotaOverhang] := m_cartRotaOverhang;
m_cartCtrlFactory[CartJointState_SlowStop] := m_cartSlowStop;

// assign controller
m_cartCtrl:=m_cartCtrlFactory[m_cartState];
m_cartCtrl.Init(m_slaveCart,m_cartCtrlCmds);
END_METHOD

METHOD PUBLIC run : BOOL
VAR_IN_OUT CONSTANT
	i_cartDataPool: ST_CartInputDataPool;
END_VAR
VAR
	i:INT;
END_VAR

// state machine transition
stateMachine(i_cartDataPool);	

//update ui data
m_slaveCart.ProcessingUIData(i_cartDataPool.m_UIData);

//update cart joint status
m_slaveCart.updateStatus();


// null ptr check
IF 0 = m_cartCtrl THEN
	RETURN;
END_IF

// run controller
m_cartCtrl.run(m_slaveCart,m_cartCtrlCmds);


m_slaveCart.updateCmds(m_cartCtrlCmds);
END_METHOD

METHOD PROTECTED stateMachine : BOOL
VAR_IN_OUT CONSTANT
	i_cartDataPool: ST_CartInputDataPool;
END_VAR
VAR
	i,j:INT;
END_VAR

// state machine transit
CASE m_cartState OF
	//cart joint error
	CartJointState_Error:
		//IF FALSE = i_cartDataPool.m_safetyData.m_slaveErrFlag THEN
		//	// to standby
		//	IF m_selfCheckPass THEN
		//		m_nextCartState :=CartJointState_Standby;
		//	ELSE
		//		m_nextCartState :=CartJointState_Init;
		//	END_IF
		//END_IF

	CartJointState_Init:
		IF m_cartCtrl.isFinished THEN
			m_nextCartState :=CartJointState_Ready;
		END_IF
		
		
	CartJointState_Ready:
		IF m_cartCtrl.isFinished  THEN
			m_nextCartState := CartJointState_InSurgery;
			
		ELSIF m_slaveCart.m_trocarOnFlag=0 AND ( i_cartDataPool.m_UIData.m_ctrlEnableFromUI.joysticks_enable OR i_cartDataPool.m_UIData.m_ctrlEnableFromUI.camera_joysticks_enable) THEN
			m_nextCartState := CartJointState_HangAdjust;
			
		ELSIF m_slaveCart.m_trocarOnFlag=0 AND (i_cartDataPool.m_UIData.m_ctrlEnableFromUI.docking_enable OR i_cartDataPool.m_UIData.m_ctrlEnableFromUI.draping_enable) THEN
			m_nextCartState := CartJointState_AsepticDeployment;
			
		ELSIF m_slaveCart.m_trocarOnFlag=0 AND  m_carHandChassisDriveUnlock[1] AND m_carHandChassisDriveUnlock[2] THEN
			m_nextCartState := CartJointState_Movement;
			
		ELSIF m_slaveCart.m_trocarOnFlag=0 AND m_slaveCart.m_rotaOverhangOnFlag > 0 THEN
			m_nextCartState := CartJointState_RotaOverhang;
		END_IF
		
	
	CartJointState_InSurgery:
		IF m_cartCtrl.isFinished  THEN
			m_nextCartState :=CartJointState_Ready;
		END_IF
		
		
	CartJointState_Movement:
		IF m_slaveCart.m_trocarOnFlag<>0 OR (NOT m_carHandChassisDriveUnlock[1] AND NOT m_carHandChassisDriveUnlock[2])  THEN
			m_nextCartState :=CartJointState_Ready;
		END_IF
		
		
	CartJointState_HangAdjust:
		IF  m_slaveCart.m_trocarOnFlag<>0 OR (NOT i_cartDataPool.m_UIData.m_ctrlEnableFromUI.joysticks_enable AND NOT i_cartDataPool.m_UIData.m_ctrlEnableFromUI.camera_joysticks_enable ) THEN
			m_nextCartState :=CartJointState_SlowStop;
		END_IF
		
		
	CartJointState_AsepticDeployment:
		IF m_cartCtrl.isFinished  THEN
			IF i_cartDataPool.m_UIData.m_ctrlEnableFromUI.docking_enable THEN
				m_slaveCart.cartDockingState := 1;
			ELSIF i_cartDataPool.m_UIData.m_ctrlEnableFromUI.draping_enable THEN
				m_slaveCart.cartDrapingState := 1;
			END_IF
			m_nextCartState :=CartJointState_Ready;
		ELSIF m_slaveCart.m_trocarOnFlag<>0 OR (NOT i_cartDataPool.m_UIData.m_ctrlEnableFromUI.docking_enable AND NOT i_cartDataPool.m_UIData.m_ctrlEnableFromUI.draping_enable) THEN
			m_nextCartState :=CartJointState_SlowStop;
		END_IF
		
		
	CartJointState_RotaOverhang:
		IF m_slaveCart.m_rotaOverhangOnFlag = 0 OR  m_slaveCart.m_trocarOnFlag<>0 THEN
			m_nextCartState :=CartJointState_SlowStop;
		END_IF
		
		
	CartJointState_SlowStop:
		IF m_cartCtrl.isFinished  THEN
			m_nextCartState :=CartJointState_Ready;
		END_IF
END_CASE

// Controller transit
IF m_nextCartState<> m_cartState THEN
	//reset current controller
	m_cartCtrl.reset();
	
	// transit to new controller
	m_lastCartState:=m_cartState;
	m_cartState:=m_nextCartState;
	m_cartCtrl:=m_cartCtrlFactory[m_cartState];
	
	//init next controller
	m_cartCtrl.Init(m_slaveCart, m_cartCtrlCmds);
	m_slaveCart.updateCmds(m_cartCtrlCmds);
END_IF
END_METHOD

END_FUNCTION_BLOCK

// ---- FBs_Robots/FB_Instrument.TcPOU
FUNCTION_BLOCK FB_Instrument

VAR_IN_OUT CONSTANT
	i_slaveArm	:FB_SlaveArm;
END_VAR

VAR
	// instrument type
	m_instruType : 	E_InstrumentType := InstruType_UNKNOWM;
	
	// flag if instrument is singer finger
	m_isSingleFinger:BOOL:= FALSE;
	
	//flag if instrument is ultrasound knife
	m_isUltrasoundKnife : BOOL := FALSE;
	
	// current and max allowed read tries
	m_curReadTries :INT :=0;
	m_maxReadTries :INT := 5;
	
	//IP of operating arm
	m_armNetId:T_AmsNetId; 	
	
	//Joint port number
	m_jointInstruAddr:UINT;	

	//Arm LED Prot	
	m_LEDPortAddr:UINT;		
	
	//The state and parameters readed from the instrument
	m_onChipData:ST_InstruOnChipData;
	
	// instrument kinematic parameters
	m_kinematicParameters:ST_InstruKinematicParam; 
	
	// joint position when instrument is at ZERO posture
	m_jntPosOffset:Vec8d;
	
	// reduction from motor joint to endoscope rotate joint
	m_endoscopeRotateReduction :LREAL := 2.0/3.0;
	
	// flag if endoscope is 30deg
	m_endoscope30Deg :BOOL:=TRUE;
	
	// udint code for zero position
	m_zeroPosCode : UDINT;
	
	// joint4 zero position, which is supposed to be a contant value
	m_jnt4ZeroPos :LREAL := 5.7;
	
	// variables used to read instrument information
	m_Step:INT;
	m_Value:UDINT;
	m_ReadDelay:TON;
	m_DealyTime:TIME:=T#0.5S;
	m_IDReadResult:UDINT;
	m_IDResult:ULINT;
	m_SeriesReadResult:UDINT;
	m_PosReadResult:UDINT;
	m_PosL1,m_PosL2,m_PosL3:UDINT;
	m_signL1,m_signL2,m_signL3:UDINT;
	m_UsageReadResult:ULINT;
	m_InstruUsageToLED:ULINT;
	m_InstruSeriesRecord:ARRAY [1..100] OF ULINT;
	m_HaveRecord:BOOL;
	m_SdoWrite:FB_EcCoESdoWrite;
	m_SdoRead:FB_EcCoESdoRead;
	
END_VAR

METHOD PROTECTED checkInstruType : BOOL
VAR_INPUT
END_VAR
VAR
	paramIdx :INT;
END_VAR
checkInstruType := m_onChipData.m_InstruID >= InstruType_First AND m_onChipData.m_InstruID <= InstruType_Last ;

// return directly if instrument ID is invalid
IF NOT(checkInstruType) THEN
	RETURN;
END_IF
m_onChipData.m_Instrutype :=  m_onChipData.m_InstruID;
m_instruType := m_onChipData.m_InstruID;
m_isSingleFinger :=  (m_instruType = InstruType_CauteryHook OR  m_instruType = InstruType_CauterySpatula );
m_isUltrasoundKnife := m_instruType = InstruType_UltrasoundKnife;

// update instrument kinematic parameters based on readed info
// TODO: move instrument kinematic parameters to chip 
paramIdx :=LIMIT(1, m_onChipData.m_InstruID, 30);
m_kinematicParameters.k13:=k13[paramIdx];
m_kinematicParameters.k23:=k23[paramIdx];
m_kinematicParameters.kx:=kx[paramIdx];
m_kinematicParameters.ky:=ky[paramIdx];
m_kinematicParameters.kz:=kz[paramIdx];
		
// rod length
IF InstruType_Endoscope =  m_instruType THEN
	m_kinematicParameters.m_rodLength := 0.48;
ELSE 
	m_kinematicParameters.m_fingerLength := 0.5392;
END_IF

// head length
IF InstruType_Endoscope =  m_instruType THEN
	m_kinematicParameters.m_headLength := 0.0;
ELSE 
	m_kinematicParameters.m_fingerLength := 0.01;
END_IF

// finger length
IF InstruType_NeedleDriver =  m_instruType THEN
	m_kinematicParameters.m_fingerLength := 0.01;
ELSE 
	m_kinematicParameters.m_fingerLength := 0.0;
END_IF

//TODO: update instrument joint motion range
IF m_isSingleFinger THEN
	m_kinematicParameters.m_wristMinDHJntPos[3]:=-110.0 * g_deg2Rad;
	m_kinematicParameters.m_wristMaxDHJntPos[3]:=110.0 * g_deg2Rad;
ELSE
	m_kinematicParameters.m_wristMinDHJntPos[3]:=-90.0 * g_deg2Rad;
	m_kinematicParameters.m_wristMaxDHJntPos[3]:=90.0 * g_deg2Rad;
END_IF
END_METHOD

PROPERTY endoscope30Deg : bool
GET
endoscope30Deg := m_endoscope30Deg;
END_GET
SET
m_endoscope30Deg := endoscope30Deg;
END_SET
END_PROPERTY

METHOD PUBLIC gripAngleMap : BOOL
VAR_INPUT
	// master gripper angle
	i_masterGripAng :LREAL;
END_VAR

VAR_OUTPUT
	// slave instrument gripper angle
	o_instruGripAngle :LREAL;
	
	// slave instrument grip force	
	o_instruGripForceLevel :LREAL;
END_VAR

VAR
	gripLevel :REAL;
END_VAR
// suppose finger is  closed and zero force if instrument has only one finger
IF m_isSingleFinger THEN
	o_instruGripAngle := 0;
	o_instruGripForceLevel:= 0;
	RETURN;
END_IF 

// finger closed and force applied
IF i_masterGripAng < g_masterGripForceStartAng THEN
	o_instruGripAngle := m_kinematicParameters.m_minGripAngle;
	// NOTE: force is applied from 50%，as minimum gripper angle already apply some sort of force
	o_instruGripForceLevel := 50+50*(g_masterGripForceStartAng - i_masterGripAng)/(g_masterGripForceStartAng - g_minMasterGripAngle);
// finger open
ELSE
	o_instruGripAngle := (g_maxMasterGripAngle - i_masterGripAng)/(g_maxMasterGripAngle - g_masterGripForceStartAng);
	o_instruGripAngle :=m_kinematicParameters.m_maxGripAngle - o_instruGripAngle * (m_kinematicParameters.m_maxGripAngle - m_kinematicParameters.m_minGripAngle);
	o_instruGripForceLevel:=0;
END_IF
END_METHOD

METHOD PROTECTED gripperAngleForwardTransform_ID12 : BOOL
VAR_INPUT
	frontAngle:LREAL;
END_VAR
VAR_OUTPUT
	endAngle:LREAL;
	Succeed:BOOL;
END_VAR
VAR
	minFrontAng :LREAL  := 16.6*2*g_deg2Rad;
	maxFrontAng :LREAL := 49.18*2*g_deg2Rad;
	AB :LREAL := 2.8;
	BC:LREAL := 5.26;
	Angle_Initial_A:LREAL := 16.6 * g_deg2Rad; 
	SIN_C,Angle_Initial_C,End_Angle_Single,Angle_Inc_C,Angle_C,SIN_A,Angle_A,Angle_Inc_A:LREAL;
END_VAR

//**************已知：器械前端开合角，求解：末端开合角***************//

//输入合法性判断，物理极限是[16.6*2，49.18*2]度
frontAngle := LIMIT(minFrontAng, frontAngle, maxFrontAng);


SIN_C:=AB*SIN(Angle_Initial_A)/BC;
Angle_Initial_C:=ASIN(SIN_C);

Angle_Inc_A:=frontAngle/2;
Angle_A:=Angle_Initial_A+Angle_Inc_A;

SIN_C:=AB*SIN(Angle_A)/BC;
Angle_C:=ASIN(SIN_C);

Angle_Inc_C:=Angle_C-Angle_Initial_C;
endAngle:=Angle_Inc_C*2;
END_METHOD

METHOD PROTECTED gripperAngleInverseTransform_ID12 : BOOL
VAR_INPUT
	endAngle:LREAL;
END_VAR
VAR_OUTPUT
	frontAngle:LREAL;
	Succeed:BOOL;
END_VAR
VAR
	minEndAng :LREAL  := 0;
	maxEndAng :LREAL := 38*g_deg2Rad;
	AB :LREAL := 2.8;
	BC:LREAL := 5.26;
	Angle_Initial_A:LREAL := 16.6 * g_deg2Rad; 
	
	SIN_C,Angle_Initial_C,End_Angle_Single,Angle_Inc_C,Angle_C,SIN_A,Angle_A,Angle_Inc_A:LREAL;
END_VAR

//***************已知：器械末端开合角，求解：前端开合角********************//

//输入合法性判断，物理极限是[0,30]度
endAngle:= LIMIT(minEndAng, endAngle, maxEndAng);

SIN_C:=AB*SIN(Angle_Initial_A)/BC;
Angle_Initial_C:=ASIN(SIN_C);

End_Angle_Single:=endAngle/2;
Angle_Inc_C:=End_Angle_Single;
Angle_C:=Angle_Initial_C+Angle_Inc_C;

SIN_A:=BC*SIN(Angle_C)/AB;
Angle_A:=ASIN(SIN_A);

Angle_Inc_A:=Angle_A-Angle_Initial_A;
frontAngle:=Angle_Inc_A*2;
END_METHOD

METHOD PUBLIC init : BOOL
VAR_INPUT
	armIdx :INT;
END_VAR
VAR
	i:INT;
END_VAR
//Update the IP and port number of the operating arm
m_armNetId:=GVL_SlaveJointEncoderCaliData.g_slaveArmNetID[armIdx];
m_jointInstruAddr:=GVL_SlaveJointEncoderCaliData.g_slaveJointNetPort[armIdx,4];

// init joint motion range
FOR i:=1 TO 3 DO
	m_kinematicParameters.m_wristMinDHJntPos[i]:=GVL_SlaveMotorParameters.g_minDHJntPos[i+3];
	m_kinematicParameters.m_wristMaxDHJntPos[i]:=GVL_SlaveMotorParameters.g_maxDHJntPos[i+3];
END_FOR
END_METHOD

METHOD PUBLIC initInstruJntPos : BOOL
VAR_INPUT
	m_curJntPos :Vec8d;
END_VAR

VAR
	i:INT;
END_VAR

FOR i := 4 TO 8 BY 1 DO
	m_jntPosOffset[i]:=m_curJntPos[i];
END_FOR
END_METHOD

// convert motor joint position to DH joint position
METHOD PUBLIC instruFK : BOOL
VAR_IN_OUT CONSTANT
	// motor joint position of slave arm
	i_jntPos :Vec8d;
END_VAR

VAR_IN_OUT
	// instrument DH  joint positon
	r_DHJntPos :Vec6d;

	// gripper angle
	r_gripAngle :LREAL;
END_VAR

VAR
	jntPosL1,jntPosL2,jntPosL3,jntPosL4,jntPosL5 :LREAL;
	gripAngle:LREAL;
END_VAR
r_DHJntPos[1]:=i_jntPos[1];
r_DHJntPos[2]:=i_jntPos[2];
r_DHJntPos[3]:=i_jntPos[3];

// ################## endoscope ############################
IF m_instruType = InstruType_endoscope THEN
	r_DHJntPos[4]:=m_endoscopeRotateReduction*(i_jntPos[8]-m_jntPosOffset[8]);
	IF m_endoscope30Deg THEN
		r_DHJntPos[5]:=-pi/2+30*g_deg2Rad;
	ELSE
		r_DHJntPos[5]:=-pi/2;
	END_IF
	r_DHJntPos[6]:=0;
	RETURN;
END_IF

//#################### instrument forward kinematic ############
// convert motor joint position to instrument joint position
jntPosL1:=(i_jntPos[4]-m_jntPosOffset[4]);
jntPosL2:=(i_jntPos[5]-m_jntPosOffset[5]);
jntPosL3:=(i_jntPos[6]-m_jntPosOffset[6]);
jntPosL4:=-(i_jntPos[7]-m_jntPosOffset[7]);
jntPosL5:=-(i_jntPos[8]-m_jntPosOffset[8]);

// diable L1 if instrument is single finger
IF m_isSingleFinger THEN
	jntPosL1 := -jntPosL2;
END_IF

// instrument FK in local coordinate
r_DHJntPos[4]:=jntPosL4/m_kinematicParameters.kx;
r_DHJntPos[5]:=jntPosL3/m_kinematicParameters.ky;
r_DHJntPos[6]:=(jntPosL1-jntPosL2-2*r_DHJntPos[5]*m_kinematicParameters.k13*m_kinematicParameters.kz)/(2*m_kinematicParameters.m_openAngleDir*m_kinematicParameters.kz);

// convert instrument rotation to arm DH joint position
r_DHJntPos[5]:=-r_DHJntPos[5]-pi/2;
r_DHJntPos[6]:=-r_DHJntPos[6];

// grip angle
gripAngle:=(jntPosL1+jntPosL2)/(m_kinematicParameters.m_openAngleDir*m_kinematicParameters.kz);



//################### gripper angle handle #################
IF (12=onChipData.m_InstruID) THEN//细齿无创抓钳
	gripperAngleForwardTransform_ID12(frontAngle:= gripAngle, endAngle=> r_gripAngle);

ELSIF (16 =onChipData.m_InstruID) THEN//单级电钩
	r_gripAngle:=0;
	
ELSIF InstruType_UltrasoundKnife = onChipData.m_InstruID THEN
	r_gripAngle:=ultrasoundKnifeGripAngleFK(jntPosL3);
	
ELSE
	r_gripAngle:=gripAngle;
END_IF
END_METHOD

METHOD PROTECTED InstruIDRecord :ARRAY [1..100] OF  ULINT
VAR_INPUT
	i_NewValue:ULINT;
	i_ArrayData:ARRAY [1..100] OF ULINT;
END_VAR

VAR
	k1:INT;
	Have_Data:BOOL;
END_VAR

FOR k1:= 1 TO 100 BY 1 DO
	IF i_NewValue=i_ArrayData[k1] THEN
		Have_Data:=TRUE;
		EXIT;
	ELSE
		Have_Data:=FALSE;
	END_IF
END_FOR

IF Have_Data=FALSE THEN
	FOR k1:= 1 TO 99 BY 1 DO
		InstruIDRecord[k1+1]:=i_ArrayData[k1];
	END_FOR
	InstruIDRecord[1]:=i_NewValue;
ELSE
	InstruIDRecord:=i_ArrayData ;
END_IF
END_METHOD

METHOD PUBLIC instruIK : BOOL
VAR_INPUT
	// DH  joint positon
	i_DHJntPos :Vec6d;

	// gripper angle
	i_gripAngle :LREAL;
	
END_VAR
VAR_OUTPUT
	o_jntPos:Vec8d;
END_VAR
VAR
	gripAngle:LREAL;
	i:INT;
	rot_x:lreal;
	rot_y:lreal;
	rot_z:lreal;

	kx,ky,kz,k13,k23:LREAL;
	open_direction:INT;
	
	d,ra:LREAL;
	AngleOffsetL3:LREAL;
	m_targetOffsetL3:LREAL;
	m_actOffsetL3:LREAL;
	
	m_gripAnglePbox:Vec8d;

	L3Offset:LREAL:=-3;
END_VAR
o_jntPos[1] := i_DHJntPos[1];
o_jntPos[2] := i_DHJntPos[2];
o_jntPos[3] := i_DHJntPos[3];

// ################## endoscope ############################
IF m_instruType = InstruType_endoscope THEN
	o_jntPos[8] := -i_DHJntPos[4]/m_endoscopeRotateReduction + m_jntPosOffset[8];
	o_jntPos[4]:=0;
	o_jntPos[5]:=0;
	o_jntPos[6]:=0;
	o_jntPos[7]:=0;
	RETURN;
END_IF

//################### gripper angle handle #################
IF (12=onChipData.m_InstruID) THEN//细齿无创抓钳
	gripperAngleInverseTransform_ID12(endAngle:= i_gripAngle, frontAngle=> gripAngle);
	
ELSIF 16 = onChipData.m_InstruID THEN//单级电钩\电铲
	gripAngle:=0;

ELSE
	gripAngle:=i_gripAngle;
END_IF

// ################# instrument inverse kinematic ##############
// convert arm DH joint position to  instrument rotation
rot_x:=i_DHJntPos[4];
rot_y:=-i_DHJntPos[5]-pi/2;
rot_z:=-i_DHJntPos[6];

// instrument IK in local coordinate
k13:=m_kinematicParameters.k13;
k23:=m_kinematicParameters.k23;
kx:=m_kinematicParameters.kx;
ky:=m_kinematicParameters.ky;
kz:=m_kinematicParameters.kz;
d:=m_kinematicParameters.m_openAngleDir;


IF InstruType_UltrasoundKnife = onChipData.m_InstruID THEN
	m_gripAnglePbox[4]:=0;
	m_gripAnglePbox[5]:=0;
	m_gripAnglePbox[6]:=ultrasoundKnifeGripAngleIK(gripAngle); 
	m_gripAnglePbox[7]:=rot_x*kx;
	m_gripAnglePbox[8]:=rot_x*kx;
ELSE
	m_gripAnglePbox[7]:=rot_x*kx;
	m_gripAnglePbox[6]:=rot_y*ky;
	ra:=gripAngle;
	m_gripAnglePbox[4]:=rot_y*k13*kz+d*rot_z*kz+d*ra*kz/2;
	m_gripAnglePbox[5]:=-rot_y*k23*kz-d*rot_z*kz+d*ra*kz/2;
END_IF

// convert instrument joint position to motor joint position
o_jntPos[4] := m_gripAnglePbox[4] + m_jntPosOffset[4];
o_jntPos[5] := m_gripAnglePbox[5] + m_jntPosOffset[5];
o_jntPos[6] := m_gripAnglePbox[6] + m_jntPosOffset[6];
o_jntPos[7] := -m_gripAnglePbox[7] + m_jntPosOffset[7];
o_jntPos[8] := -m_gripAnglePbox[8] + m_jntPosOffset[8];
END_METHOD

// convert motor joint velocity to DH joint velocity
METHOD PUBLIC instruJntVelFK : BOOL
VAR_IN_OUT CONSTANT
	// motor joint velocity of slave arm
	i_jntVel :Vec8d;
END_VAR

VAR_IN_OUT
	// instrument DH  joint velocity
	r_DHJntVel :Vec6d;
END_VAR

VAR
	jntPosL1,jntPosL2,jntPosL3,jntPosL4,jntPosL5 :LREAL;
	gripAngle:LREAL;
END_VAR
r_DHJntVel[1]:=i_jntVel[1];
r_DHJntVel[2]:=i_jntVel[2];
r_DHJntVel[3]:=i_jntVel[3];

r_DHJntVel[4]:=-i_jntVel[7]/m_kinematicParameters.kx;
r_DHJntVel[5]:=i_jntVel[6]/m_kinematicParameters.ky;
r_DHJntVel[6]:=(i_jntVel[4]-i_jntVel[5]-2*r_DHJntVel[5]*m_kinematicParameters.k13*m_kinematicParameters.kz)/(2*m_kinematicParameters.m_openAngleDir*m_kinematicParameters.kz);
r_DHJntVel[5]:=-r_DHJntVel[5];
r_DHJntVel[6]:=-r_DHJntVel[6];
END_METHOD

METHOD PROTECTED InstruSreiesFind : BOOL
VAR_INPUT
	i_NewValue:ULINT;
	i_ArrayData:ARRAY [1..100] OF ULINT;
	
END_VAR

VAR
	k1:INT;
END_VAR
InstruSreiesFind:=FALSE;
FOR k1:= 1 TO 100 BY 1 DO
	IF i_NewValue=i_ArrayData[k1] THEN
		InstruSreiesFind:=TRUE;
		EXIT;
	ELSE
		InstruSreiesFind:=FALSE;
	END_IF
END_FOR
END_METHOD

PROPERTY kinematicParameters :REFERENCE TO ST_InstruKinematicParam
GET
kinematicParameters ref=m_kinematicParameters;
END_GET
END_PROPERTY

PROPERTY onChipData : REFERENCE TO ST_InstruOnChipData
GET
onChipData ref=m_onChipData;
END_GET
END_PROPERTY

METHOD PUBLIC readParameters : BOOL
VAR_INPUT
	startFlag :BOOL;
END_VAR

VAR
	paramIdx :INT;
END_VAR
// TODO: read m_kinematic parameters from chip 
//Take the rising edge of the read signal
m_ReadDelay(IN:= m_Step=10, PT:= m_DealyTime, Q=> , ET=> );//计时器
IF startFlag AND m_curReadTries < m_maxReadTries THEN
	m_Step:=0;
	m_onChipData.m_InstruReadSucceed:=FALSE;
	m_onChipData.m_Error:=FALSE;
	m_onChipData.m_ErrorID:=0;
END_IF


CASE m_Step OF
	
	0://向6093发送0x8000  0000---发送读取信号
		m_Value:=16#80000000; 
		m_SdoWrite(sNetId:= m_ArmNetId, nSlaveAddr:= m_JointInstruAddr, nSubIndex:= 0, nIndex:= 16#6093, pSrcBuf:= ADR(m_Value), cbBufLen:= SIZEOF(m_Value), bExecute:= TRUE, );
		IF NOT m_SdoWrite.bBusy THEN
			m_SdoWrite(bExecute:=FALSE);
			m_Step:=10;
		END_IF
		
		
	10://延时0.5s、防止值还没有返回
		IF m_ReadDelay.Q THEN
			m_Step:=20;
		END_IF

		
	20://从6093地址中拿值
		m_SdoRead(sNetId:= m_ArmNetId, nSlaveAddr:= m_JointInstruAddr,	nSubIndex:= 0, nIndex:= 16#6093, pDstBuf:= ADR(m_IDReadResult), cbBufLen:= SIZEOF(m_IDReadResult), bExecute:= TRUE, 	tTimeout:= , bBusy=> , bError=> , nErrId=> , cbRead=> );
		IF NOT m_SdoRead.bBusy THEN
			m_SdoRead(bExecute:=FALSE);
			m_Step:=30;
		END_IF	
		
	
	30://处理器械ID、低16位
		m_IDResult:=UDINT_TO_ULINT(16#0000FFFF AND m_IDReadResult);
		m_Step:=40;
		
		
	40://读取6095、器械序列号
		m_SdoRead(sNetId:= m_ArmNetId, nSlaveAddr:= m_JointInstruAddr,	nSubIndex:= 0, nIndex:= 16#6095, pDstBuf:= ADR(m_SeriesReadResult), cbBufLen:= SIZEOF(m_SeriesReadResult), bExecute:= TRUE, 	tTimeout:= , bBusy=> , bError=> , nErrId=> , cbRead=> );
		IF NOT m_SdoRead.bBusy THEN
			m_SdoRead(bExecute:=FALSE);
			m_Step:=50;
		END_IF	
	
		
	50://处理序列号，低30位
		m_onChipData.m_InstruseriesNum:=SHL(m_IDResult,31)+(16#7FFFFFFF AND m_SeriesReadResult);
		m_onChipData.m_InstruID:=LREAL_TO_INT(FLOOR(lr_in:= m_onChipData.m_InstruseriesNum/EXPT(10,9))); //取十进制前三位为器械ID
		m_Step:=60;
		
		
	60://读取6096---器械零点位置
		m_SdoRead(sNetId:= m_ArmNetId, nSlaveAddr:= m_JointInstruAddr,	nSubIndex:= 0, nIndex:= 16#6096, pDstBuf:= ADR(m_PosReadResult), cbBufLen:= SIZEOF(m_PosReadResult), bExecute:= TRUE, 	tTimeout:= , bBusy=> , bError=> , nErrId=> , cbRead=> );
		IF NOT m_SdoRead.bBusy THEN
			m_SdoRead(bExecute:=FALSE);
			m_Step:=70;
		END_IF	
		
		
	70: //处理位置，L1:0-9位，L2:10-19位，L3:20-29位
		zeroPosDecode(m_PosReadResult, o_q1=>m_onChipData.m_InstruPos[1],o_q2=>m_onChipData.m_InstruPos[2],o_q3=>m_onChipData.m_InstruPos[3]);
		m_onChipData.m_InstruPos[4] := m_jnt4ZeroPos;
		m_onChipData.m_InstruPos[5] := 0;
		
		m_Step:=80;
		
	80://读取器械使用次数 6094
		m_SdoRead(sNetId:= m_ArmNetId, nSlaveAddr:= m_JointInstruAddr,	nSubIndex:= 0, nIndex:= 16#6094, pDstBuf:= ADR(m_UsageReadResult), cbBufLen:= SIZEOF(m_UsageReadResult), bExecute:= TRUE, 	tTimeout:= , bBusy=> , bError=> , nErrId=> , cbRead=> );
		IF NOT m_SdoRead.bBusy THEN
			m_SdoRead(bExecute:=FALSE);
			m_Step:=90;
		END_IF	
		
		
	90://处理器械使用次数读取结果
		m_onChipData.m_InstruusageCounts:=m_UsageReadResult;
		m_InstruUsageToLED:=LIMIT(0,m_UsageReadResult,99);
		m_Step:=110;
		
		
	100://将器械使用次数写入LED
		m_Value:=ULINT_TO_UDINT(16#FFFF AND m_InstruUsageToLED) ;
		m_SdoWrite(sNetId:= m_ArmNetId, nSlaveAddr:= m_LEDPortAddr, nSubIndex:= 06, nIndex:= 16#6090, pSrcBuf:= ADR(m_Value), cbBufLen:= SIZEOF(m_Value), bExecute:= TRUE, tTimeout:= , bBusy=> , bError=> , nErrId=> );
		IF NOT m_SdoWrite.bBusy THEN
			m_SdoWrite(bExecute:=FALSE);
			m_Step:=110;
		END_IF
		
	110://处理当器械使用次数达到上限后、在同一场手术中还能使用
		IF m_onChipData.m_InstruusageCounts=m_onChipData.m_InstrumaxUsageCounts THEN
			m_InstruSeriesRecord:=InstruIDRecord(i_NewValue:= m_onChipData.m_InstruusageCounts, i_ArrayData:= m_InstruSeriesRecord);
			m_Step:=120;
		ELSE
			m_Step:=120;
		END_IF
		
		
	120://结果诊断
		m_onChipData.m_InstruReadSucceed:=checkInstruType();
		IF NOT(m_onChipData.m_InstruReadSucceed) THEN
			m_onChipData.m_Error:=TRUE;
			m_onChipData.m_ErrorID:=1;
(*		ELSIF m_onChipData.m_InstruusageCounts>m_onChipData.m_InstrumaxUsageCounts AND m_onChipData.m_InstruID<>20 THEN
			m_HaveRecord:=InstruSreiesFind(i_NewValue:=m_onChipData.m_InstruseriesNum , i_ArrayData:=m_InstruSeriesRecord );
			IF m_HaveRecord THEN
				m_onChipData.m_Instrutype:=2;
				m_onChipData.m_InstruReadSucceed:=TRUE;
				m_Step:=130;
			ELSE
				m_onChipData.m_Error:=TRUE;
				m_onChipData.m_ErrorID:=2;
			END_IF*)
		END_IF
		m_Step :=-1;
		m_curReadTries := m_curReadTries +1;
	
END_CASE
END_METHOD

METHOD PUBLIC reset : BOOL
VAR_INPUT
END_VAR
VAR
	i:INT;
END_VAR
m_Step := -1;
m_curReadTries := 0;
m_onChipData.m_InstruID := 0;
m_onChipData.m_InstruseriesNum :=0;
m_onChipData.m_Instrutype :=InstruType_UNKNOWM;
m_onChipData.m_Error:=FALSE;
m_onChipData.m_ErrorID:=0;
m_onChipData.m_InstruReadSucceed:=FALSE;
m_isSingleFinger:=FALSE;
m_instruType:=InstruType_UNKNOWM;

FOR i:= 4 TO 8 BY 1 DO
	m_jntPosOffset[i]:=0;
END_FOR

// init joint motion range
FOR i:=1 TO 3 DO
	m_kinematicParameters.m_wristMinDHJntPos[i]:=GVL_SlaveMotorParameters.g_minDHJntPos[i+3];
	m_kinematicParameters.m_wristMaxDHJntPos[i]:=GVL_SlaveMotorParameters.g_maxDHJntPos[i+3];
END_FOR
END_METHOD

METHOD ultrasoundKnifeGripAngleFK : LREAL
VAR_IN_OUT CONSTANT
	// motor joint position of slave arm
	i_jntPos :LREAL;
END_VAR

VAR
	m_jntPos : LREAL;
END_VAR

m_jntPos := i_jntPos;

m_jntPos := LIMIT (-20*g_deg2Rad,m_jntPos,70*g_deg2Rad);

ultrasoundKnifeGripAngleFK := ASIN((m_jntPos*g_uknifeMotorLead * g_uknifeLeverRatio/(2*pi) -  g_uknifeGripTravel * SIN(g_uknifeGripDividAngle))/g_uknifeGripTravel)+g_uknifeGripDividAngle;
END_METHOD

METHOD ultrasoundKnifeGripAngleIK : LREAL
VAR_INPUT
	// gripper angle
	i_gripAngle :LREAL;
END_VAR

VAR
	m_gripAngle : LREAL;
END_VAR

m_gripAngle := i_gripAngle;

ultrasoundKnifeGripAngleIK := (g_uknifeGripTravel * (SIN(g_uknifeGripDividAngle) - SIN(g_uknifeGripDividAngle - m_gripAngle))/(g_uknifeMotorLead*g_uknifeLeverRatio/(2*pi)));
END_METHOD

METHOD PUBLIC writeZeroPosToChip : BOOL
VAR_INPUT
	i_q1:LREAL;
	i_q2:LREAL;
	i_q3:LREAL;
END_VAR
zeroPosCode(i_q1,i_q2,i_q3, o_code=>m_zeroPosCode);

writeZeroPosToChip:=FALSE;
m_SdoWrite(sNetId:= m_ArmNetId, nSlaveAddr:= m_JointInstruAddr, nSubIndex:= 0, nIndex:= 16#6096, pSrcBuf:= ADR(m_zeroPosCode), cbBufLen:= SIZEOF(m_zeroPosCode), bExecute:= TRUE, );
IF NOT m_SdoWrite.bBusy THEN
	m_SdoWrite(bExecute:=FALSE);
	writeZeroPosToChip:=TRUE;
END_IF
END_METHOD

// code instrument joints(4/5/6) zero position as a UDINT
// joint1 : bit 21-30; joint2: bit 11-20; joint3: bit1-10
// zeroPos: [0, 2pi]; code:[0-3sFF]
METHOD PROTECTED zeroPosCode : BOOL
VAR_INPUT
	i_q1:LREAL;
	i_q2:LREAL;
	i_q3:LREAL;
END_VAR
VAR_OUTPUT
	o_code:UDINT;
END_VAR
VAR
	posCode:UDINT;
END_VAR
// highest bit set to 1
o_code:=2;

// joint1
posCode := LREAL_TO_UDINT(16#3FF * LIMIT(0,i_q1/g_2pi,1));
o_code := SHL(o_code, 10);
o_code := o_code OR posCode;

// joint2
posCode := LREAL_TO_UDINT(16#3FF * LIMIT(0,i_q2/g_2pi,1));
o_code := SHL(o_code, 10);
o_code := o_code OR posCode;

// joint3
posCode := LREAL_TO_UDINT(16#3FF * LIMIT(0,i_q3/g_2pi,1));
o_code := SHL(o_code, 10);
o_code := o_code OR posCode;
END_METHOD

// decode instrument joints(4/5/6) zero position from a UDINT
// joint1 : bit 21-30; joint2: bit 11-20; joint4: bit1-10
// zeroPos: [0, 2pi]; code:[0-2FF]
METHOD PROTECTED zeroPosDecode : BOOL
VAR_INPUT
	i_posCode :UDINT;
END_VAR
VAR_OUTPUT
	o_q1:LREAL;
	o_q2:LREAL;
	o_q3:LREAL;
END_VAR
VAR
	posCode:UDINT;
END_VAR
// joint3
posCode := i_posCode AND 16#3FF;
o_q3 := g_2pi *  posCode/16#3FF;

// joint2
i_posCode := SHR(i_posCode, 10);
posCode := i_posCode AND 16#3FF;
o_q2 := g_2pi *  posCode/16#3FF;

// joint1
i_posCode := SHR(i_posCode, 10);
posCode := i_posCode AND 16#3FF;
o_q1 := g_2pi *  posCode/16#3FF;
END_METHOD

END_FUNCTION_BLOCK

// ---- FBs_Robots/FB_SlaveJoint.TcPOU
FUNCTION_BLOCK FB_SlaveJoint EXTENDS FB_JointBase
VAR_INPUT
END_VAR
VAR_OUTPUT
END_VAR
VAR
	// power box joint motor rated current
	m_wristJntRatedCurrent : DINT := 200;

END_VAR

METHOD PUBLIC init : BOOL
VAR_INPUT
	i_armIdx :INT;
	i_jntIdx :INT;
	i_controlCycleTime :LREAL;
	// velocity is calculated every (m_velCalcCycles) control cycles
	// TODO: insturment joint motor can not reach 4k now, so calculate their velocity with 1k frequency, need to remove later
	i_velCalcCycles :INT;
END_VAR
m_armIdx:=i_armIdx;
m_jntIdx:=i_jntIdx;
m_cycleTime := i_controlCycleTime;
m_velCalcCycles :=MAX(i_velCalcCycles,1);

// hardware parameters
m_motorEncoderRes :=GVL_SlaveMotorParameters.g_incEncoderRes[i_jntIdx];
m_linkEncoderRes :=GVL_SlaveMotorParameters.g_absEncoderRes[i_jntIdx];
m_motorReduction :=GVL_SlaveMotorParameters.g_motorReduction[i_jntIdx];
m_linkEncoderReduction :=GVL_SlaveMotorParameters.g_absEncoderReduction[i_jntIdx];
m_trqConst :=GVL_SlaveMotorParameters.g_motorTrqConst[i_jntIdx];
m_maxCurrent :=GVL_SlaveMotorParameters.g_motorMaxCurrent[i_jntIdx];
m_motorDir :=GVL_SlaveMotorParameters.g_motorDir[i_jntIdx];								
m_minJntPos	:=GVL_SlaveMotorParameters.g_minJntPos[i_jntIdx];
m_maxJntPos	:=GVL_SlaveMotorParameters.g_maxJntPos[i_jntIdx];

//link encoder calibartion data
m_linkEncoderDir :=GVL_SlaveJointEncoderCaliData.g_asbEncoderDir[i_jntIdx];
m_minLinkEncoder :=GVL_SlaveJointEncoderCaliData.g_minLinkEncoder[i_armIdx, i_jntIdx] - m_linkEncoderDir*GVL_SlaveJointEncoderCaliData.g_linkEncLimitBuffer; // expand limit
m_maxLinkEncoder :=GVL_SlaveJointEncoderCaliData.g_maxLinkEncoder[i_armIdx, i_jntIdx] + m_linkEncoderDir*GVL_SlaveJointEncoderCaliData.g_linkEncLimitBuffer; // expand limit
m_caliLinkEncoder :=GVL_SlaveJointEncoderCaliData.g_caliLinkEncoder[i_armIdx, i_jntIdx];
m_linkEncCaliJntPos :=GVL_SlaveJointEncoderCaliData.g_linkEncCaliJntPos[i_jntIdx];
m_linkEncZeroCross :=GVL_SlaveJointEncoderCaliData.g_linkEncZeroCross[i_armIdx, i_jntIdx];
m_multiCycles :=GVL_SlaveJointEncoderCaliData.g_multipleCyclesJoint[i_armIdx,i_jntIdx];

// convert cali link encoder if joint cross zero
IF 1=m_linkEncZeroCross THEN
	IF 1=m_linkEncoderDir AND m_caliLinkEncoder < m_minLinkEncoder THEN
		m_caliLinkEncoder := GVL_SlaveJointEncoderCaliData.g_caliLinkEncoder[i_armIdx, i_jntIdx] + m_linkEncoderRes;
	ELSIF -1=m_linkEncoderDir AND m_caliLinkEncoder < m_maxLinkEncoder THEN
		m_caliLinkEncoder := GVL_SlaveJointEncoderCaliData.g_caliLinkEncoder[i_armIdx, i_jntIdx] + m_linkEncoderRes;
	END_IF
END_IF

// macro data
m_trq2CurrentRatio:=m_motorDir * 1000.0/(m_trqConst*m_motorReduction);
m_current2TrqRatio:=m_motorDir * (m_trqConst*m_motorReduction)/1000.0;
m_linkEnc2PosRatio := 2*PI*m_linkEncoderDir/(m_linkEncoderReduction*m_linkEncoderRes);
m_motorEnc2PosRatio := 2*PI * m_motorDir/(m_motorReduction * m_motorEncoderRes);

// motor data init
m_rawJntVel :=0;
m_curJntVel:=0;
m_curJntTrq :=0;
m_rawCurrent :=0;
m_filtCurrent :=0;
m_cmdJntVel :=0.0;
m_cmdJntTrq :=0.0;
m_cmdCurrent := 0.0;

// filter init
m_jntVelLpf.init(1, GVL_SlaveControlParameters.g_curJntVelLpfCutoffFreq, g_slaveArmCtrlFreq/m_velCalcCycles);
m_cmdTrqLpf.init(1, GVL_SlaveControlParameters.g_cmdJntTrqLpfCutoffFreq, g_slaveArmCtrlFreq);
m_curTrqLpf.init(1, GVL_SlaveControlParameters.g_curJntTrqLpfCutoffFreq, g_slaveArmCtrlFreq);

// driver init value
m_motorOutputs.m_controlWord:=DriverCtrlWord_INIT;
m_motorOutputs.m_opMode:=INT_TO_SINT(DriverOPMode_Pos);
m_motorOutputs.m_cmdCurrent:=0;
m_motorOutputs.m_cmdMotorEncoder:=m_motorInputs.m_motorEncoder;
END_METHOD

METHOD PUBLIC updateCmds : BOOL
VAR_INPUT
	i_opMode : E_DriverOPMode;
	i_cmdPos :LREAL;
	i_cmdTrq :LREAL;
END_VAR
VAR
	filtCmdTrq :LREAL;
END_VAR
SUPER^.updateCmds(i_opMode, i_cmdPos, i_cmdTrq);

// write SDO data
//writeSDOData();
END_METHOD

METHOD PROTECTED writeSDOData : BOOL
VAR_INPUT
END_VAR
VAR
	SDOSubIndexMode :WORD;
	SDOSubIndexCur :WORD;
END_VAR
//动力盒移动关节和器械旋转关节，共享一个控制字，由SDO写入
IF (m_jntIdx=3) OR (m_jntIdx=8)  THEN
	SDOSubIndexMode :=16#609B;
	SDOSubIndexCur:=16#6098;
//动力盒3、5号电机为一个驱动器，共享一个控制字，由SDO写入
ELSIF (m_jntIdx=4) OR (m_jntIdx=6)  THEN
	SDOSubIndexMode :=16#609C;
	SDOSubIndexCur:=16#6099;
//动力盒2、4号电机为一个驱动器，共享一个控制字，由SDO写入
ELSIF (m_jntIdx=5) OR (m_jntIdx=7)  THEN
	SDOSubIndexMode :=16#609D;
	SDOSubIndexCur:=16#609A;
END_IF

IF m_jntIdx <3 THEN
	RETURN;
END_IF

// write driver operation mode if it changs
IF  m_jntIdx >=3 AND m_jntIdx <=7 THEN
	m_opModeSDOWrite(sNetID:= GVL_SlaveJointEncoderCaliData.g_slaveArmNetID[m_armIdx],
					nSlaveAddr := GVL_SlaveJointEncoderCaliData.g_slaveJointNetPort[m_armIdx,m_jntIdx],
					nSubIndex:=0,nIndex:=SDOSubIndexMode,pSrcBuf:=ADR(m_motorOutputs.m_opMode),cbBufLen:=SIZEOF(m_motorOutputs.m_opMode),bExecute:=TRUE);
	IF NOT m_opModeSDOWrite.bBusy THEN
		m_opModeSDOWrite(bExecute:=FALSE);
	END_IF
END_IF

// write max motor current if it changes and works in position mode
IF m_jntIdx >=4 AND m_jntIdx <=8  THEN 
	m_MotorCurrentSDOWrite(sNetID:= GVL_SlaveJointEncoderCaliData.g_slaveArmNetID[m_armIdx],
					nSlaveAddr := GVL_SlaveJointEncoderCaliData.g_slaveJointNetPort[m_armIdx,m_jntIdx],
					nSubIndex:=0,nIndex:=SDOSubIndexCur,pSrcBuf:=ADR(m_wristJntRatedCurrent),cbBufLen:=SIZEOF(m_wristJntRatedCurrent),bExecute:=TRUE);
	IF NOT m_MotorCurrentSDOWrite.bBusy THEN
		m_MotorCurrentSDOWrite(bExecute:=FALSE);
	END_IF
END_IF
END_METHOD

END_FUNCTION_BLOCK

// ---- FBs_SetupControllers/FB_SetupCtrlJnt5GraCali.TcPOU
// Brief: setup arm gravity calibration
// For trajectory synchronizaiton, the planner generate a trajecotry for setup joint3/5 and slave joint 1-3, but only former used here 
FUNCTION_BLOCK PUBLIC FB_SetupCtrlJnt5GraCali EXTENDS FB_SetupArmCtrlBase
VAR_INPUT
END_VAR
VAR_OUTPUT
END_VAR
VAR
// cali trajectory
	m_caliMotionSegs :INT :=3;
	m_graCaliTraj:ARRAY [1..3] OF LREAL:=[PI/2-pi/3, PI/2-PI/6, PI/2-pi/3];
	
		 
	m_caliMaxjntVel:LREAL:=2.5 * g_deg2Rad;
	m_caliMaxjntAcc:LREAL:=0.5;
	m_caliMaxjntJerk:LREAL:=2.0;
	
	m_caliTrajIdx: INT := 1;
	m_caliPlanner: ARRAY[1..3] OF FB_BasicDoubleS;
	
END_VAR

// override this function in each exact controller
METHOD PROTECTED calcCmdJntPos : BOOL
VAR_IN_OUT CONSTANT
	i_setupArm	:FB_SetupArm;
END_VAR


VAR 
	i :INT;
	curJntVel :Vec5d;
END_VAR
// safety check
IF ABS(i_setupArm.curJntVel[5]) > 10*g_deg2Rad THEN
	m_isFinished:=TRUE;
	RETURN;
END_IF

// check if planner is ready
IF m_caliPlanner[m_caliTrajIdx].isGene = FALSE THEN
	calcCmdJntPos:=FALSE;
	RETURN;
END_IF

// traj plan
calcCmdJntPos :=m_caliPlanner[m_caliTrajIdx].evaluate(m_timePeriod, q=> m_cmdJntPos[5], q_dot=>m_cmdJntVel[5], q_ddot=> m_cmdJntAcc[5]);

// check if to transit to next segment
IF(m_timePeriod > m_caliPlanner[m_caliTrajIdx].duration  AND ABS(i_setupArm.curJntVel[5])<GVL_SlaveControlParameters.g_jntStaticVelThres) THEN
	m_caliTrajIdx:=m_caliTrajIdx+1;
	m_timePeriod:=0;
END_IF

// check if to terminated
IF(m_caliTrajIdx > m_caliMotionSegs) THEN
	m_isFinished:=TRUE;
END_IF
END_METHOD

METHOD PUBLIC init : BOOL
VAR_IN_OUT CONSTANT
	i_setupArm	:FB_SetupArm;
END_VAR
VAR_IN_OUT 
	r_setupArmCtrlCmd :ST_SetupArmCtrlCmds;
END_VAR

VAR
	i,j :INT;
	startJntPos,endJntPos :LREAL;
	q,v:ARRAY[1..2] OF lreal;
END_VAR
SUPER^.Init(i_setupArm,r_setupArmCtrlCmd);
m_jntEnableFlag[5]:=1;
m_jntOPMode[5]:= DriverOPMode_PosTrq;
m_caliTrajIdx :=1;

// traj plan
// fisrt segment
q[1]:=i_setupArm.curJntPos[5];
q[2]:=m_graCaliTraj[1];
v[1]:=0;
v[2]:=0;
m_caliPlanner[1].init(q,v,m_caliMaxjntVel, m_caliMaxJntAcc, m_caliMaxJntJerk);

// other segments
FOR i:=2 TO m_caliMotionSegs DO 
	q[1]:=m_graCaliTraj[i-1];
	q[2]:=m_graCaliTraj[i];
	m_caliPlanner[i].init(q,v,m_caliMaxjntVel, m_caliMaxJntAcc, m_caliMaxJntJerk);
END_FOR
END_METHOD

END_FUNCTION_BLOCK

// ---- FBs_SetupControllers/FB_SetupCtrlManualAdjust.TcPOU
// Brief: Setup Arm Adjust
FUNCTION_BLOCK PUBLIC FB_SetupCtrlManualAdjust EXTENDS FB_SetupArmCtrlBase
VAR_INPUT
END_VAR
VAR_OUTPUT
END_VAR
VAR
	// friction compensation scale
	m_frictionScale :LREAL :=0.5;
	
	// velocity threshold for friction compensation 
	m_jnt3FrictionCompVelLow :LREAL := 0.0005;
	m_frictionScaleLow :LREAL :=0.3;
	m_jnt3FrictionCompVelMiddle :LREAL := 0.005;
	m_frictionScaleMiddle :LREAL :=0.5;
	m_jnt3FrictionCompVelHigh :LREAL := 0.05;
	m_frictionScaleHigh :LREAL :=0.7;
	
	// jnt5 adjust velocity
	m_jnt5MaxAdjustVel :LREAL:=5.0*g_deg2Rad;
	m_jnt5MaxAdjustAcc :LREAL:=60*g_deg2Rad;
	
	// jnt5 enabled time period
	m_jnt5EnableTime :LREAL :=0;
	
	// time threshold to drive jnt5 after it's enabled
	m_jnt5AdjustWaitTime :LREAL := 0.25;

END_VAR

// override this function in each exact controller
METHOD PROTECTED calcCmdJntPos : BOOL
VAR_IN_OUT CONSTANT
	i_setupArm	:FB_SetupArm;
END_VAR


